   DATA[2120,25] := 2.0;
   DATA[2120,26] := 7.873174;
   DATA[2120,27] := 144.322;
   DATA[2120,28] := 262.0161;
   DATA[2120,29] := 12.03538;
   DATA[2120,30] := 1.726096;
   DATA[2120,31] := 1.28372;
   DATA[2120,32] := 0.7353967;
   DATA[2120,33] := 0.3084265;
   DATA[2120,34] := 2.0;
   DATA[2120,35] := 250.1122;
   DATA[2120,36] := 1.69801;
   DATA[2120,37] := 189.0381;
   DATA[2120,38] := 0.000128152;
   DATA[2120,39] := 1.0;
   DATA[2120,40] := 1.0;
   DATA[2121,0] := 2.573103;
   DATA[2121,1] := 862.3046;
   DATA[2121,2] := 2.0;
   DATA[2121,3] := 2.0;
   DATA[2121,4] := 262.4007;
   DATA[2121,5] := 8.392271;
   DATA[2121,6] := 330.7357;
   DATA[2121,7] := 2.461667;
   DATA[2121,8] := 2.0;
   DATA[2121,9] := 2.0;
   DATA[2121,10] := 2.0;
   DATA[2121,11] := 19.72598;
   DATA[2121,12] := 2.209013;
   DATA[2121,13] := 806.564;
   DATA[2121,14] := 1.0;
   DATA[2121,15] := 2.0;
   DATA[2121,16] := 1.0;
   DATA[2121,17] := 1.0;
   DATA[2121,18] := 1.0;
   DATA[2121,19] := 2.0;
   DATA[2121,20] := 148.808;
   DATA[2121,21] := 154.8065;
   DATA[2121,22] := 1.717489;
   DATA[2121,23] := 839.131;
   DATA[2121,24] := 2.0;
   DATA[2121,25] := 2.0;
   DATA[2121,26] := 7.873174;
   DATA[2121,27] := 144.322;
   DATA[2121,28] := 262.0161;
   DATA[2121,29] := 12.03538;
   DATA[2121,30] := 1.725968;
   DATA[2121,31] := 1.300884;
   DATA[2121,32] := 0.7353967;
   DATA[2121,33] := 0.3084265;
   DATA[2121,34] := 2.0;
   DATA[2121,35] := 250.1122;
   DATA[2121,36] := 1.69801;
   DATA[2121,37] := 189.0381;
   DATA[2121,38] := 0.000128152;
   DATA[2121,39] := 1.0;
   DATA[2121,40] := 1.0;
   DATA[2122,0] := 2.608013;
   DATA[2122,1] := 862.6971;
   DATA[2122,2] := 2.0;
   DATA[2122,3] := 2.0;
   DATA[2122,4] := 262.4007;
   DATA[2122,5] := 8.392271;
   DATA[2122,6] := 330.7357;
   DATA[2122,7] := 2.461667;
   DATA[2122,8] := 2.0;
   DATA[2122,9] := 2.0;
   DATA[2122,10] := 2.0;
   DATA[2122,11] := 19.67155;
   DATA[2122,12] := 2.209013;
   DATA[2122,13] := 806.3237;
   DATA[2122,14] := 1.0;
   DATA[2122,15] := 2.0;
   DATA[2122,16] := 1.0;
   DATA[2122,17] := 1.0;
   DATA[2122,18] := 1.0;
   DATA[2122,19] := 2.0;
   DATA[2122,20] := 148.808;
   DATA[2122,21] := 154.8065;
   DATA[2122,22] := 1.719156;
   DATA[2122,23] := 839.2463;
   DATA[2122,24] := 2.0;
   DATA[2122,25] := 2.0;
   DATA[2122,26] := 7.873174;
   DATA[2122,27] := 144.322;
   DATA[2122,28] := 262.0161;
   DATA[2122,29] := 12.03538;
   DATA[2122,30] := 1.725968;
   DATA[2122,31] := 1.30178;
   DATA[2122,32] := 0.7353967;
   DATA[2122,33] := 0.3084265;
   DATA[2122,34] := 2.0;
   DATA[2122,35] := 250.3365;
   DATA[2122,36] := 1.69801;
   DATA[2122,37] := 189.0381;
   DATA[2122,38] := 0.000128152;
   DATA[2122,39] := 1.0;
   DATA[2122,40] := 1.0;
   DATA[2123,0] := 2.641322;
   DATA[2123,1] := 862.3831;
   DATA[2123,2] := 2.0;
   DATA[2123,3] := 2.0;
   DATA[2123,4] := 262.4007;
   DATA[2123,5] := 8.392271;
   DATA[2123,6] := 330.787;
   DATA[2123,7] := 2.461667;
   DATA[2123,8] := 2.0;
   DATA[2123,9] := 2.0;
   DATA[2123,10] := 2.0;
   DATA[2123,11] := 19.66835;
   DATA[2123,12] := 2.209013;
   DATA[2123,13] := 806.4038;
   DATA[2123,14] := 1.0;
   DATA[2123,15] := 2.0;
   DATA[2123,16] := 1.0;
   DATA[2123,17] := 1.0;
   DATA[2123,18] := 1.0;
   DATA[2123,19] := 2.0;
   DATA[2123,20] := 148.808;
   DATA[2123,21] := 154.8065;
   DATA[2123,22] := 1.719156;
   DATA[2123,23] := 839.0541;
   DATA[2123,24] := 2.0;
   DATA[2123,25] := 2.0;
   DATA[2123,26] := 7.873174;
   DATA[2123,27] := 144.322;
   DATA[2123,28] := 262.0161;
   DATA[2123,29] := 12.03538;
   DATA[2123,30] := 1.725968;
   DATA[2123,31] := 1.30178;
   DATA[2123,32] := 0.7353967;
   DATA[2123,33] := 0.3084265;
   DATA[2123,34] := 2.0;
   DATA[2123,35] := 250.3365;
   DATA[2123,36] := 1.69801;
   DATA[2123,37] := 189.0381;
   DATA[2123,38] := 0.000128152;
   DATA[2123,39] := 1.0;
   DATA[2123,40] := 1.0;
   DATA[2124,0] := 2.660539;
   DATA[2124,1] := 862.6971;
   DATA[2124,2] := 2.0;
   DATA[2124,3] := 2.0;
   DATA[2124,4] := 262.4007;
   DATA[2124,5] := 8.392271;
   DATA[2124,6] := 330.787;
   DATA[2124,7] := 2.461667;
   DATA[2124,8] := 2.0;
   DATA[2124,9] := 2.0;
   DATA[2124,10] := 2.0;
   DATA[2124,11] := 19.64594;
   DATA[2124,12] := 2.212087;
   DATA[2124,13] := 806.524;
   DATA[2124,14] := 1.0;
   DATA[2124,15] := 2.0;
   DATA[2124,16] := 1.0;
   DATA[2124,17] := 1.0;
   DATA[2124,18] := 1.0;
   DATA[2124,19] := 2.0;
   DATA[2124,20] := 148.808;
   DATA[2124,21] := 154.8065;
   DATA[2124,22] := 1.719156;
   DATA[2124,23] := 839.131;
   DATA[2124,24] := 2.0;
   DATA[2124,25] := 2.0;
   DATA[2124,26] := 7.873174;
   DATA[2124,27] := 144.322;
   DATA[2124,28] := 262.0161;
   DATA[2124,29] := 12.03538;
   DATA[2124,30] := 1.725968;
   DATA[2124,31] := 1.29243;
   DATA[2124,32] := 0.7353967;
   DATA[2124,33] := 0.3084265;
   DATA[2124,34] := 2.0;
   DATA[2124,35] := 250.3365;
   DATA[2124,36] := 1.69801;
   DATA[2124,37] := 189.0861;
   DATA[2124,38] := 0.000128152;
   DATA[2124,39] := 1.0;
   DATA[2124,40] := 1.0;
   DATA[2125,0] := 2.660539;
   DATA[2125,1] := 862.8934;
   DATA[2125,2] := 2.0;
   DATA[2125,3] := 2.0;
   DATA[2125,4] := 262.4007;
   DATA[2125,5] := 8.392271;
   DATA[2125,6] := 330.787;
   DATA[2125,7] := 2.461667;
   DATA[2125,8] := 2.0;
   DATA[2125,9] := 2.0;
   DATA[2125,10] := 2.0;
   DATA[2125,11] := 19.64594;
   DATA[2125,12] := 2.212087;
   DATA[2125,13] := 806.524;
   DATA[2125,14] := 1.0;
   DATA[2125,15] := 2.0;
   DATA[2125,16] := 1.0;
   DATA[2125,17] := 1.0;
   DATA[2125,18] := 1.0;
   DATA[2125,19] := 2.0;
   DATA[2125,20] := 148.808;
   DATA[2125,21] := 154.8065;
   DATA[2125,22] := 1.717874;
   DATA[2125,23] := 839.2079;
   DATA[2125,24] := 2.0;
   DATA[2125,25] := 2.0;
   DATA[2125,26] := 7.874135;
   DATA[2125,27] := 144.322;
   DATA[2125,28] := 262.0161;
   DATA[2125,29] := 12.03538;
   DATA[2125,30] := 1.725968;
   DATA[2125,31] := 1.276419;
   DATA[2125,32] := 0.7353967;
   DATA[2125,33] := 0.3084265;
   DATA[2125,34] := 2.0;
   DATA[2125,35] := 250.3365;
   DATA[2125,36] := 1.69801;
   DATA[2125,37] := 189.1662;
   DATA[2125,38] := 0.000128152;
   DATA[2125,39] := 1.0;
   DATA[2125,40] := 1.0;
   DATA[2126,0] := 2.641642;
   DATA[2126,1] := 863.0897;
   DATA[2126,2] := 2.0;
   DATA[2126,3] := 2.0;
   DATA[2126,4] := 262.4007;
   DATA[2126,5] := 8.392271;
   DATA[2126,6] := 330.8383;
   DATA[2126,7] := 2.461282;
   DATA[2126,8] := 2.0;
   DATA[2126,9] := 2.0;
   DATA[2126,10] := 2.0;
   DATA[2126,11] := 19.64594;
   DATA[2126,12] := 2.212087;
   DATA[2126,13] := 806.6842;
   DATA[2126,14] := 1.0;
   DATA[2126,15] := 2.0;
   DATA[2126,16] := 1.0;
   DATA[2126,17] := 1.0;
   DATA[2126,18] := 1.0;
   DATA[2126,19] := 2.0;
   DATA[2126,20] := 148.808;
   DATA[2126,21] := 154.8065;
   DATA[2126,22] := 1.716849;
   DATA[2126,23] := 839.5924;
   DATA[2126,24] := 2.0;
   DATA[2126,25] := 2.0;
   DATA[2126,26] := 7.874135;
   DATA[2126,27] := 144.322;
   DATA[2126,28] := 262.0161;
   DATA[2126,29] := 12.03538;
   DATA[2126,30] := 1.725968;
   DATA[2126,31] := 1.271295;
   DATA[2126,32] := 0.7353967;
   DATA[2126,33] := 0.3084265;
   DATA[2126,34] := 2.0;
   DATA[2126,35] := 250.3365;
   DATA[2126,36] := 1.69801;
   DATA[2126,37] := 189.1662;
   DATA[2126,38] := 0.000128152;
   DATA[2126,39] := 1.0;
   DATA[2126,40] := 1.0;
   DATA[2127,0] := 2.630433;
   DATA[2127,1] := 862.8934;
   DATA[2127,2] := 2.0;
   DATA[2127,3] := 2.0;
   DATA[2127,4] := 262.4007;
   DATA[2127,5] := 8.392271;
   DATA[2127,6] := 330.8383;
   DATA[2127,7] := 2.458847;
   DATA[2127,8] := 2.0;
   DATA[2127,9] := 2.0;
   DATA[2127,10] := 2.0;
   DATA[2127,11] := 19.70677;
   DATA[2127,12] := 2.212087;
   DATA[2127,13] := 806.2036;
   DATA[2127,14] := 1.0;
   DATA[2127,15] := 2.0;
   DATA[2127,16] := 1.0;
   DATA[2127,17] := 1.0;
   DATA[2127,18] := 1.0;
   DATA[2127,19] := 2.0;
   DATA[2127,20] := 148.808;
   DATA[2127,21] := 154.8065;
   DATA[2127,22] := 1.716849;
   DATA[2127,23] := 839.4771;
   DATA[2127,24] := 2.0;
   DATA[2127,25] := 2.0;
   DATA[2127,26] := 7.874135;
   DATA[2127,27] := 144.322;
   DATA[2127,28] := 262.0161;
   DATA[2127,29] := 12.03538;
   DATA[2127,30] := 1.72789;
   DATA[2127,31] := 1.277443;
   DATA[2127,32] := 0.7353967;
   DATA[2127,33] := 0.3084265;
   DATA[2127,34] := 2.0;
   DATA[2127,35] := 250.3365;
   DATA[2127,36] := 1.69801;
   DATA[2127,37] := 189.1662;
   DATA[2127,38] := 0.000128152;
   DATA[2127,39] := 1.0;
   DATA[2127,40] := 1.0;
   DATA[2128,0] := 2.623387;
   DATA[2128,1] := 863.2859;
   DATA[2128,2] := 2.0;
   DATA[2128,3] := 2.0;
   DATA[2128,4] := 262.4007;
   DATA[2128,5] := 8.392271;
   DATA[2128,6] := 330.8383;
   DATA[2128,7] := 2.458847;
   DATA[2128,8] := 2.0;
   DATA[2128,9] := 2.0;
   DATA[2128,10] := 2.0;
   DATA[2128,11] := 19.70677;
   DATA[2128,12] := 2.210294;
   DATA[2128,13] := 806.524;
   DATA[2128,14] := 1.0;
   DATA[2128,15] := 2.0;
   DATA[2128,16] := 1.0;
   DATA[2128,17] := 1.0;
   DATA[2128,18] := 1.0;
   DATA[2128,19] := 2.0;
   DATA[2128,20] := 148.808;
   DATA[2128,21] := 154.8065;
   DATA[2128,22] := 1.716849;
   DATA[2128,23] := 839.5155;
   DATA[2128,24] := 2.0;
   DATA[2128,25] := 2.0;
   DATA[2128,26] := 7.874135;
   DATA[2128,27] := 144.322;
   DATA[2128,28] := 262.0161;
   DATA[2128,29] := 12.03538;
   DATA[2128,30] := 1.728275;
   DATA[2128,31] := 1.291277;
   DATA[2128,32] := 0.7353967;
   DATA[2128,33] := 0.3084265;
   DATA[2128,34] := 2.0;
   DATA[2128,35] := 250.3365;
   DATA[2128,36] := 1.69801;
   DATA[2128,37] := 189.1662;
   DATA[2128,38] := 0.000128152;
   DATA[2128,39] := 1.0;
   DATA[2128,40] := 1.0;
   DATA[2129,0] := 2.622105;
   DATA[2129,1] := 862.9719;
   DATA[2129,2] := 2.0;
   DATA[2129,3] := 2.0;
   DATA[2129,4] := 262.4007;
   DATA[2129,5] := 8.392271;
   DATA[2129,6] := 330.8383;
   DATA[2129,7] := 2.458078;
   DATA[2129,8] := 2.0;
   DATA[2129,9] := 2.0;
   DATA[2129,10] := 2.0;
   DATA[2129,11] := 19.73558;
   DATA[2129,12] := 2.209269;
   DATA[2129,13] := 805.9232;
   DATA[2129,14] := 1.0;
   DATA[2129,15] := 2.0;
   DATA[2129,16] := 1.0;
   DATA[2129,17] := 1.0;
   DATA[2129,18] := 1.0;
   DATA[2129,19] := 2.0;
   DATA[2129,20] := 148.808;
   DATA[2129,21] := 154.8065;
   DATA[2129,22] := 1.716849;
   DATA[2129,23] := 839.2463;
   DATA[2129,24] := 2.0;
   DATA[2129,25] := 2.0;
   DATA[2129,26] := 7.874135;
   DATA[2129,27] := 144.322;
   DATA[2129,28] := 262.0161;
   DATA[2129,29] := 12.03538;
   DATA[2129,30] := 1.728275;
   DATA[2129,31] := 1.291789;
   DATA[2129,32] := 0.7353967;
   DATA[2129,33] := 0.3084265;
   DATA[2129,34] := 2.0;
   DATA[2129,35] := 250.3365;
   DATA[2129,36] := 1.69801;
   DATA[2129,37] := 189.1662;
   DATA[2129,38] := 0.000128152;
   DATA[2129,39] := 1.0;
   DATA[2129,40] := 1.0;
   DATA[2130,0] := 2.606091;
   DATA[2130,1] := 863.2859;
   DATA[2130,2] := 2.0;
   DATA[2130,3] := 2.0;
   DATA[2130,4] := 262.4007;
   DATA[2130,5] := 8.392271;
   DATA[2130,6] := 330.8383;
   DATA[2130,7] := 2.458078;
   DATA[2130,8] := 2.0;
   DATA[2130,9] := 2.0;
   DATA[2130,10] := 2.0;
   DATA[2130,11] := 19.73558;
   DATA[2130,12] := 2.209269;
   DATA[2130,13] := 805.9232;
   DATA[2130,14] := 1.0;
   DATA[2130,15] := 2.0;
   DATA[2130,16] := 1.0;
   DATA[2130,17] := 1.0;
   DATA[2130,18] := 1.0;
   DATA[2130,19] := 2.0;
   DATA[2130,20] := 148.808;
   DATA[2130,21] := 154.8065;
   DATA[2130,22] := 1.716849;
   DATA[2130,23] := 839.4001;
   DATA[2130,24] := 2.0;
   DATA[2130,25] := 2.0;
   DATA[2130,26] := 7.874135;
   DATA[2130,27] := 144.322;
   DATA[2130,28] := 262.0161;
   DATA[2130,29] := 12.03538;
   DATA[2130,30] := 1.728275;
   DATA[2130,31] := 1.289868;
   DATA[2130,32] := 0.7379573;
   DATA[2130,33] := 0.3084265;
   DATA[2130,34] := 2.0;
   DATA[2130,35] := 250.3365;
   DATA[2130,36] := 1.69801;
   DATA[2130,37] := 189.1662;
   DATA[2130,38] := 0.000128152;
   DATA[2130,39] := 1.0;
   DATA[2130,40] := 1.0;
   DATA[2131,0] := 2.587195;
   DATA[2131,1] := 863.5999;
   DATA[2131,2] := 2.0;
   DATA[2131,3] := 2.0;
   DATA[2131,4] := 262.4007;
   DATA[2131,5] := 8.392271;
   DATA[2131,6] := 330.8383;
   DATA[2131,7] := 2.458078;
   DATA[2131,8] := 2.0;
   DATA[2131,9] := 2.0;
   DATA[2131,10] := 2.0;
   DATA[2131,11] := 19.77079;
   DATA[2131,12] := 2.209269;
   DATA[2131,13] := 805.7229;
   DATA[2131,14] := 1.0;
   DATA[2131,15] := 2.0;
   DATA[2131,16] := 1.0;
   DATA[2131,17] := 1.0;
   DATA[2131,18] := 1.0;
   DATA[2131,19] := 2.0;
   DATA[2131,20] := 148.808;
   DATA[2131,21] := 154.8065;
   DATA[2131,22] := 1.716849;
   DATA[2131,23] := 839.0541;
   DATA[2131,24] := 2.0;
   DATA[2131,25] := 2.0;
   DATA[2131,26] := 7.874135;
   DATA[2131,27] := 144.322;
   DATA[2131,28] := 262.0161;
   DATA[2131,29] := 12.03538;
   DATA[2131,30] := 1.726096;
   DATA[2131,31] := 1.269117;
   DATA[2131,32] := 0.7379573;
   DATA[2131,33] := 0.3084265;
   DATA[2131,34] := 2.0;
   DATA[2131,35] := 250.3365;
   DATA[2131,36] := 1.69801;
   DATA[2131,37] := 189.1662;
   DATA[2131,38] := 0.000128152;
   DATA[2131,39] := 1.0;
   DATA[2131,40] := 1.0;
   DATA[2132,0] := 2.567338;
   DATA[2132,1] := 863.4822;
   DATA[2132,2] := 2.0;
   DATA[2132,3] := 2.0;
   DATA[2132,4] := 262.4007;
   DATA[2132,5] := 8.392271;
   DATA[2132,6] := 330.8383;
   DATA[2132,7] := 2.458078;
   DATA[2132,8] := 2.0;
   DATA[2132,9] := 2.0;
   DATA[2132,10] := 2.0;
   DATA[2132,11] := 19.77079;
   DATA[2132,12] := 2.209269;
   DATA[2132,13] := 805.8831;
   DATA[2132,14] := 1.0;
   DATA[2132,15] := 2.0;
   DATA[2132,16] := 1.0;
   DATA[2132,17] := 1.0;
   DATA[2132,18] := 1.0;
   DATA[2132,19] := 2.0;
   DATA[2132,20] := 148.808;
   DATA[2132,21] := 154.8065;
   DATA[2132,22] := 1.717746;
   DATA[2132,23] := 839.3232;
   DATA[2132,24] := 2.0;
   DATA[2132,25] := 2.0;
   DATA[2132,26] := 7.874135;
   DATA[2132,27] := 144.322;
   DATA[2132,28] := 262.0161;
   DATA[2132,29] := 12.03538;
   DATA[2132,30] := 1.726096;
   DATA[2132,31] := 1.265659;
   DATA[2132,32] := 0.7379573;
   DATA[2132,33] := 0.3084265;
   DATA[2132,34] := 2.0;
   DATA[2132,35] := 250.4326;
   DATA[2132,36] := 1.69801;
   DATA[2132,37] := 189.1662;
   DATA[2132,38] := 0.000128152;
   DATA[2132,39] := 1.0;
   DATA[2132,40] := 1.0;
   DATA[2133,0] := 2.558691;
   DATA[2133,1] := 863.8354;
   DATA[2133,2] := 2.0;
   DATA[2133,3] := 2.0;
   DATA[2133,4] := 262.4007;
   DATA[2133,5] := 8.392271;
   DATA[2133,6] := 330.8383;
   DATA[2133,7] := 2.458078;
   DATA[2133,8] := 2.0;
   DATA[2133,9] := 2.0;
   DATA[2133,10] := 2.0;
   DATA[2133,11] := 19.77079;
   DATA[2133,12] := 2.209269;
   DATA[2133,13] := 805.7229;
   DATA[2133,14] := 1.0;
   DATA[2133,15] := 2.0;
   DATA[2133,16] := 1.0;
   DATA[2133,17] := 1.0;
   DATA[2133,18] := 1.0;
   DATA[2133,19] := 2.0;
   DATA[2133,20] := 148.808;
   DATA[2133,21] := 154.9603;
   DATA[2133,22] := 1.718771;
   DATA[2133,23] := 839.0541;
   DATA[2133,24] := 2.0;
   DATA[2133,25] := 2.0;
   DATA[2133,26] := 7.874135;
   DATA[2133,27] := 144.322;
   DATA[2133,28] := 262.0161;
   DATA[2133,29] := 12.03538;
   DATA[2133,30] := 1.726096;
   DATA[2133,31] := 1.280902;
   DATA[2133,32] := 0.7366771;
   DATA[2133,33] := 0.3070813;
   DATA[2133,34] := 2.0;
   DATA[2133,35] := 250.4967;
   DATA[2133,36] := 1.69801;
   DATA[2133,37] := 189.1662;
   DATA[2133,38] := 0.000128152;
   DATA[2133,39] := 1.0;
   DATA[2133,40] := 1.0;
   DATA[2134,0] := 2.535951;
   DATA[2134,1] := 863.7962;
   DATA[2134,2] := 2.0;
   DATA[2134,3] := 2.0;
   DATA[2134,4] := 262.4007;
   DATA[2134,5] := 8.392271;
   DATA[2134,6] := 330.8383;
   DATA[2134,7] := 2.458078;
   DATA[2134,8] := 2.0;
   DATA[2134,9] := 2.0;
   DATA[2134,10] := 2.0;
   DATA[2134,11] := 19.77079;
   DATA[2134,12] := 2.209269;
   DATA[2134,13] := 805.6829;
   DATA[2134,14] := 1.0;
   DATA[2134,15] := 2.0;
   DATA[2134,16] := 1.0;
   DATA[2134,17] := 1.0;
   DATA[2134,18] := 1.0;
   DATA[2134,19] := 2.0;
   DATA[2134,20] := 148.808;
   DATA[2134,21] := 154.9603;
   DATA[2134,22] := 1.718771;
   DATA[2134,23] := 839.2463;
   DATA[2134,24] := 2.0;
   DATA[2134,25] := 2.0;
   DATA[2134,26] := 7.874135;
   DATA[2134,27] := 144.322;
   DATA[2134,28] := 262.0161;
   DATA[2134,29] := 12.03538;
   DATA[2134,30] := 1.726096;
   DATA[2134,31] := 1.280005;
   DATA[2134,32] := 0.7359089;
   DATA[2134,33] := 0.3070813;
   DATA[2134,34] := 2.0;
   DATA[2134,35] := 250.4967;
   DATA[2134,36] := 1.69801;
   DATA[2134,37] := 189.1662;
   DATA[2134,38] := 0.000128152;
   DATA[2134,39] := 1.0;
   DATA[2134,40] := 1.0;
   DATA[2135,0] := 2.520257;
   DATA[2135,1] := 864.1887;
   DATA[2135,2] := 2.0;
   DATA[2135,3] := 2.0;
   DATA[2135,4] := 262.4007;
   DATA[2135,5] := 8.392271;
   DATA[2135,6] := 330.8383;
   DATA[2135,7] := 2.459744;
   DATA[2135,8] := 2.0;
   DATA[2135,9] := 2.0;
   DATA[2135,10] := 2.0;
   DATA[2135,11] := 19.73238;
   DATA[2135,12] := 2.209269;
   DATA[2135,13] := 805.5627;
   DATA[2135,14] := 1.0;
   DATA[2135,15] := 2.0;
   DATA[2135,16] := 1.0;
   DATA[2135,17] := 1.0;
   DATA[2135,18] := 1.0;
   DATA[2135,19] := 2.0;
   DATA[2135,20] := 148.808;
   DATA[2135,21] := 154.9603;
   DATA[2135,22] := 1.720309;
   DATA[2135,23] := 838.8234;
   DATA[2135,24] := 2.0;
   DATA[2135,25] := 2.0;
   DATA[2135,26] := 7.874135;
   DATA[2135,27] := 144.322;
   DATA[2135,28] := 262.0161;
   DATA[2135,29] := 12.03538;
   DATA[2135,30] := 1.726096;
   DATA[2135,31] := 1.275778;
   DATA[2135,32] := 0.7348846;
   DATA[2135,33] := 0.3075297;
   DATA[2135,34] := 2.0;
   DATA[2135,35] := 250.4967;
   DATA[2135,36] := 1.69801;
   DATA[2135,37] := 189.2143;
   DATA[2135,38] := 0.000128152;
   DATA[2135,39] := 1.0;
   DATA[2135,40] := 1.0;
   DATA[2136,0] := 2.502642;
   DATA[2136,1] := 864.385;
   DATA[2136,2] := 2.0;
   DATA[2136,3] := 2.0;
   DATA[2136,4] := 262.4007;
   DATA[2136,5] := 8.392271;
   DATA[2136,6] := 330.8383;
   DATA[2136,7] := 2.459744;
   DATA[2136,8] := 2.0;
   DATA[2136,9] := 2.0;
   DATA[2136,10] := 2.0;
   DATA[2136,11] := 19.73238;
   DATA[2136,12] := 2.209269;
   DATA[2136,13] := 805.4025;
   DATA[2136,14] := 1.0;
   DATA[2136,15] := 2.0;
   DATA[2136,16] := 1.0;
   DATA[2136,17] := 1.0;
   DATA[2136,18] := 1.0;
   DATA[2136,19] := 2.0;
   DATA[2136,20] := 148.808;
   DATA[2136,21] := 154.9603;
   DATA[2136,22] := 1.720309;
   DATA[2136,23] := 838.6311;
   DATA[2136,24] := 2.0;
   DATA[2136,25] := 2.0;
   DATA[2136,26] := 7.874135;
   DATA[2136,27] := 144.322;
   DATA[2136,28] := 262.0161;
   DATA[2136,29] := 12.03538;
   DATA[2136,30] := 1.726096;
   DATA[2136,31] := 1.276419;
   DATA[2136,32] := 0.7348846;
   DATA[2136,33] := 0.3083624;
   DATA[2136,34] := 2.0;
   DATA[2136,35] := 250.4967;
   DATA[2136,36] := 1.69801;
   DATA[2136,37] := 189.3585;
   DATA[2136,38] := 0.000128152;
   DATA[2136,39] := 1.0;
   DATA[2136,40] := 1.0;
   DATA[2137,0] := 2.48823;
   DATA[2137,1] := 864.6205;
   DATA[2137,2] := 2.0;
   DATA[2137,3] := 2.0;
   DATA[2137,4] := 262.4007;
   DATA[2137,5] := 8.392271;
   DATA[2137,6] := 330.8126;
   DATA[2137,7] := 2.460129;
   DATA[2137,8] := 2.0;
   DATA[2137,9] := 2.0;
   DATA[2137,10] := 2.0;
   DATA[2137,11] := 19.73238;
   DATA[2137,12] := 2.209269;
   DATA[2137,13] := 805.2022;
   DATA[2137,14] := 1.0;
   DATA[2137,15] := 2.0;
   DATA[2137,16] := 1.0;
   DATA[2137,17] := 1.0;
   DATA[2137,18] := 1.0;
   DATA[2137,19] := 2.0;
   DATA[2137,20] := 148.808;
   DATA[2137,21] := 154.9603;
   DATA[2137,22] := 1.720309;
   DATA[2137,23] := 838.0928;
   DATA[2137,24] := 2.0;
   DATA[2137,25] := 2.0;
   DATA[2137,26] := 7.874135;
   DATA[2137,27] := 144.322;
   DATA[2137,28] := 262.0161;
   DATA[2137,29] := 12.03538;
   DATA[2137,30] := 1.728019;
   DATA[2137,31] := 1.270398;
   DATA[2137,32] := 0.7348846;
   DATA[2137,33] := 0.3075937;
   DATA[2137,34] := 2.0;
   DATA[2137,35] := 250.4967;
   DATA[2137,36] := 1.69801;
   DATA[2137,37] := 189.3585;
   DATA[2137,38] := 0.000128152;
   DATA[2137,39] := 1.0;
   DATA[2137,40] := 1.0;
   DATA[2138,0] := 2.467092;
   DATA[2138,1] := 864.8168;
   DATA[2138,2] := 2.0;
   DATA[2138,3] := 2.0;
   DATA[2138,4] := 262.4007;
   DATA[2138,5] := 8.392271;
   DATA[2138,6] := 330.6075;
   DATA[2138,7] := 2.460129;
   DATA[2138,8] := 2.0;
   DATA[2138,9] := 2.0;
   DATA[2138,10] := 2.0;
   DATA[2138,11] := 19.73238;
   DATA[2138,12] := 2.210037;
   DATA[2138,13] := 805.3224;
   DATA[2138,14] := 1.0;
   DATA[2138,15] := 2.0;
   DATA[2138,16] := 1.0;
   DATA[2138,17] := 1.0;
   DATA[2138,18] := 1.0;
   DATA[2138,19] := 2.0;
   DATA[2138,20] := 148.808;
   DATA[2138,21] := 154.9603;
   DATA[2138,22] := 1.720309;
   DATA[2138,23] := 838.1312;
   DATA[2138,24] := 2.0;
   DATA[2138,25] := 2.0;
   DATA[2138,26] := 7.874135;
   DATA[2138,27] := 144.322;
   DATA[2138,28] := 262.0161;
   DATA[2138,29] := 12.03538;
   DATA[2138,30] := 1.728788;
   DATA[2138,31] := 1.278468;
   DATA[2138,32] := 0.7348846;
   DATA[2138,33] := 0.3069532;
   DATA[2138,34] := 2.0;
   DATA[2138,35] := 250.4967;
   DATA[2138,36] := 1.69801;
   DATA[2138,37] := 189.3585;
   DATA[2138,38] := 0.000128152;
   DATA[2138,39] := 1.0;
   DATA[2138,40] := 1.0;
   DATA[2139,0] := 2.458764;
   DATA[2139,1] := 864.6597;
   DATA[2139,2] := 2.0;
   DATA[2139,3] := 2.0;
   DATA[2139,4] := 262.4007;
   DATA[2139,5] := 8.392271;
   DATA[2139,6] := 330.6075;
   DATA[2139,7] := 2.460129;
   DATA[2139,8] := 2.0;
   DATA[2139,9] := 2.0;
   DATA[2139,10] := 2.0;
   DATA[2139,11] := 19.73238;
   DATA[2139,12] := 2.21055;
   DATA[2139,13] := 805.2022;
   DATA[2139,14] := 1.0;
   DATA[2139,15] := 2.0;
   DATA[2139,16] := 1.0;
   DATA[2139,17] := 1.0;
   DATA[2139,18] := 1.0;
   DATA[2139,19] := 2.0;
   DATA[2139,20] := 148.808;
   DATA[2139,21] := 155.0884;
   DATA[2139,22] := 1.720309;
   DATA[2139,23] := 838.0928;
   DATA[2139,24] := 2.0;
   DATA[2139,25] := 2.0;
   DATA[2139,26] := 7.874135;
   DATA[2139,27] := 144.322;
   DATA[2139,28] := 262.0161;
   DATA[2139,29] := 12.03538;
   DATA[2139,30] := 1.728788;
   DATA[2139,31] := 1.296016;
   DATA[2139,32] := 0.7348846;
   DATA[2139,33] := 0.3065048;
   DATA[2139,34] := 2.0;
   DATA[2139,35] := 250.4967;
   DATA[2139,36] := 1.69801;
   DATA[2139,37] := 189.3585;
   DATA[2139,38] := 0.000128152;
   DATA[2139,39] := 1.0;
   DATA[2139,40] := 1.0;
   DATA[2140,0] := 2.436665;
   DATA[2140,1] := 864.4635;
   DATA[2140,2] := 2.0;
   DATA[2140,3] := 2.0;
   DATA[2140,4] := 262.4007;
   DATA[2140,5] := 8.392271;
   DATA[2140,6] := 330.6075;
   DATA[2140,7] := 2.460641;
   DATA[2140,8] := 2.0;
   DATA[2140,9] := 2.0;
   DATA[2140,10] := 2.0;
   DATA[2140,11] := 19.7836;
   DATA[2140,12] := 2.21055;
   DATA[2140,13] := 804.6815;
   DATA[2140,14] := 1.0;
   DATA[2140,15] := 2.0;
   DATA[2140,16] := 1.0;
   DATA[2140,17] := 1.0;
   DATA[2140,18] := 1.0;
   DATA[2140,19] := 2.0;
   DATA[2140,20] := 148.808;
   DATA[2140,21] := 155.0884;
   DATA[2140,22] := 1.720309;
   DATA[2140,23] := 837.7852;
   DATA[2140,24] := 2.0;
   DATA[2140,25] := 2.0;
   DATA[2140,26] := 7.874135;
   DATA[2140,27] := 144.322;
   DATA[2140,28] := 262.0161;
   DATA[2140,29] := 12.03538;
   DATA[2140,30] := 1.728788;
   DATA[2140,31] := 1.310747;
   DATA[2140,32] := 0.7348846;
   DATA[2140,33] := 0.3065048;
   DATA[2140,34] := 2.0;
   DATA[2140,35] := 250.4967;
   DATA[2140,36] := 1.69801;
   DATA[2140,37] := 189.2464;
   DATA[2140,38] := 0.000128152;
   DATA[2140,39] := 1.0;
   DATA[2140,40] := 1.0;
   DATA[2141,0] := 2.428018;
   DATA[2141,1] := 864.228;
   DATA[2141,2] := 2.0;
   DATA[2141,3] := 2.0;
   DATA[2141,4] := 262.4007;
   DATA[2141,5] := 8.392271;
   DATA[2141,6] := 330.6075;
   DATA[2141,7] := 2.462564;
   DATA[2141,8] := 2.0;
   DATA[2141,9] := 2.0;
   DATA[2141,10] := 2.0;
   DATA[2141,11] := 19.7836;
   DATA[2141,12] := 2.21055;
   DATA[2141,13] := 804.6014;
   DATA[2141,14] := 1.0;
   DATA[2141,15] := 2.0;
   DATA[2141,16] := 1.0;
   DATA[2141,17] := 1.0;
   DATA[2141,18] := 1.0;
   DATA[2141,19] := 2.0;
   DATA[2141,20] := 148.808;
   DATA[2141,21] := 155.0884;
   DATA[2141,22] := 1.716464;
   DATA[2141,23] := 838.0543;
   DATA[2141,24] := 2.0;
   DATA[2141,25] := 2.0;
   DATA[2141,26] := 7.874135;
   DATA[2141,27] := 144.322;
   DATA[2141,28] := 262.0161;
   DATA[2141,29] := 12.03538;
   DATA[2141,30] := 1.728788;
   DATA[2141,31] := 1.312284;
   DATA[2141,32] := 0.7348846;
   DATA[2141,33] := 0.3065048;
   DATA[2141,34] := 2.0;
   DATA[2141,35] := 250.4967;
   DATA[2141,36] := 1.69801;
   DATA[2141,37] := 189.2464;
   DATA[2141,38] := 0.000128152;
   DATA[2141,39] := 1.0;
   DATA[2141,40] := 1.0;
   DATA[2142,0] := 2.428018;
   DATA[2142,1] := 864.2672;
   DATA[2142,2] := 2.0;
   DATA[2142,3] := 2.0;
   DATA[2142,4] := 262.4007;
   DATA[2142,5] := 8.392271;
   DATA[2142,6] := 330.6075;
   DATA[2142,7] := 2.463845;
   DATA[2142,8] := 2.0;
   DATA[2142,9] := 2.0;
   DATA[2142,10] := 2.0;
   DATA[2142,11] := 19.7836;
   DATA[2142,12] := 2.209525;
   DATA[2142,13] := 804.8017;
   DATA[2142,14] := 1.0;
   DATA[2142,15] := 2.0;
   DATA[2142,16] := 1.0;
   DATA[2142,17] := 1.0;
   DATA[2142,18] := 1.0;
   DATA[2142,19] := 2.0;
   DATA[2142,20] := 148.808;
   DATA[2142,21] := 155.0884;
   DATA[2142,22] := 1.716464;
   DATA[2142,23] := 838.4773;
   DATA[2142,24] := 2.0;
   DATA[2142,25] := 2.0;
   DATA[2142,26] := 7.874135;
   DATA[2142,27] := 144.1938;
   DATA[2142,28] := 262.0161;
   DATA[2142,29] := 12.03538;
   DATA[2142,30] := 1.728788;
   DATA[2142,31] := 1.308569;
   DATA[2142,32] := 0.7348846;
   DATA[2142,33] := 0.3065048;
   DATA[2142,34] := 2.0;
   DATA[2142,35] := 250.3525;
   DATA[2142,36] := 1.69801;
   DATA[2142,37] := 189.2464;
   DATA[2142,38] := 0.000128152;
   DATA[2142,39] := 1.0;
   DATA[2142,40] := 1.0;
   DATA[2143,0] := 2.43058;
   DATA[2143,1] := 864.385;
   DATA[2143,2] := 2.0;
   DATA[2143,3] := 2.0;
   DATA[2143,4] := 262.4007;
   DATA[2143,5] := 8.392271;
   DATA[2143,6] := 330.6075;
   DATA[2143,7] := 2.463845;
   DATA[2143,8] := 2.0;
   DATA[2143,9] := 2.0;
   DATA[2143,10] := 2.0;
   DATA[2143,11] := 19.7836;
   DATA[2143,12] := 2.209397;
   DATA[2143,13] := 804.5613;
   DATA[2143,14] := 1.0;
   DATA[2143,15] := 2.0;
   DATA[2143,16] := 1.0;
   DATA[2143,17] := 1.0;
   DATA[2143,18] := 1.0;
   DATA[2143,19] := 2.0;
   DATA[2143,20] := 148.808;
   DATA[2143,21] := 155.0884;
   DATA[2143,22] := 1.716464;
   DATA[2143,23] := 838.6311;
   DATA[2143,24] := 2.0;
   DATA[2143,25] := 2.0;
   DATA[2143,26] := 7.874135;
   DATA[2143,27] := 144.1938;
   DATA[2143,28] := 262.0161;
   DATA[2143,29] := 12.03538;
   DATA[2143,30] := 1.726737;
   DATA[2143,31] := 1.288715;
   DATA[2143,32] := 0.7348846;
   DATA[2143,33] := 0.3065048;
   DATA[2143,34] := 2.0;
   DATA[2143,35] := 250.3525;
   DATA[2143,36] := 1.69801;
   DATA[2143,37] := 189.2464;
   DATA[2143,38] := 0.000128152;
   DATA[2143,39] := 1.0;
   DATA[2143,40] := 1.0;
   DATA[2144,0] := 2.466771;
   DATA[2144,1] := 864.2672;
   DATA[2144,2] := 2.0;
   DATA[2144,3] := 2.0;
   DATA[2144,4] := 262.4007;
   DATA[2144,5] := 8.392271;
   DATA[2144,6] := 330.6075;
   DATA[2144,7] := 2.462564;
   DATA[2144,8] := 2.0;
   DATA[2144,9] := 2.0;
   DATA[2144,10] := 2.0;
   DATA[2144,11] := 19.64594;
   DATA[2144,12] := 2.209397;
   DATA[2144,13] := 804.8017;
   DATA[2144,14] := 1.0;
   DATA[2144,15] := 2.0;
   DATA[2144,16] := 1.0;
   DATA[2144,17] := 1.0;
   DATA[2144,18] := 1.0;
   DATA[2144,19] := 2.0;
   DATA[2144,20] := 148.808;
   DATA[2144,21] := 155.0884;
   DATA[2144,22] := 1.713261;
   DATA[2144,23] := 839.0925;
   DATA[2144,24] := 2.0;
   DATA[2144,25] := 2.0;
   DATA[2144,26] := 7.874135;
   DATA[2144,27] := 144.1938;
   DATA[2144,28] := 262.0161;
   DATA[2144,29] := 12.03538;
   DATA[2144,30] := 1.72507;
   DATA[2144,31] := 1.281927;
   DATA[2144,32] := 0.7348846;
   DATA[2144,33] := 0.3065048;
   DATA[2144,34] := 2.0;
   DATA[2144,35] := 250.3525;
   DATA[2144,36] := 1.69801;
   DATA[2144,37] := 188.974;
   DATA[2144,38] := 0.000128152;
   DATA[2144,39] := 1.0;
   DATA[2144,40] := 1.0;
   DATA[2145,0] := 2.513532;
   DATA[2145,1] := 864.071;
   DATA[2145,2] := 2.0;
   DATA[2145,3] := 2.0;
   DATA[2145,4] := 262.4007;
   DATA[2145,5] := 8.392271;
   DATA[2145,6] := 330.6075;
   DATA[2145,7] := 2.462179;
   DATA[2145,8] := 2.0;
   DATA[2145,9] := 2.0;
   DATA[2145,10] := 2.0;
   DATA[2145,11] := 19.56591;
   DATA[2145,12] := 2.209397;
   DATA[2145,13] := 805.002;
   DATA[2145,14] := 1.0;
   DATA[2145,15] := 2.0;
   DATA[2145,16] := 1.0;
   DATA[2145,17] := 1.0;
   DATA[2145,18] := 1.0;
   DATA[2145,19] := 2.0;
   DATA[2145,20] := 148.808;
   DATA[2145,21] := 155.0884;
   DATA[2145,22] := 1.713261;
   DATA[2145,23] := 838.9387;
   DATA[2145,24] := 2.0;
   DATA[2145,25] := 2.0;
   DATA[2145,26] := 7.874135;
   DATA[2145,27] := 144.1938;
   DATA[2145,28] := 262.0161;
   DATA[2145,29] := 12.03538;
   DATA[2145,30] := 1.72507;
   DATA[2145,31] := 1.271935;
   DATA[2145,32] := 0.7353967;
   DATA[2145,33] := 0.3065048;
   DATA[2145,34] := 2.0;
   DATA[2145,35] := 250.2403;
   DATA[2145,36] := 1.69801;
   DATA[2145,37] := 188.974;
   DATA[2145,38] := 0.000128152;
   DATA[2145,39] := 1.0;
   DATA[2145,40] := 1.0;
   DATA[2146,0] := 2.550364;
   DATA[2146,1] := 863.8354;
   DATA[2146,2] := 2.0;
   DATA[2146,3] := 2.0;
   DATA[2146,4] := 262.4007;
   DATA[2146,5] := 8.392271;
   DATA[2146,6] := 330.6075;
   DATA[2146,7] := 2.461667;
   DATA[2146,8] := 2.0;
   DATA[2146,9] := 2.0;
   DATA[2146,10] := 2.0;
   DATA[2146,11] := 19.50829;
   DATA[2146,12] := 2.209397;
   DATA[2146,13] := 805.5226;
   DATA[2146,14] := 1.0;
   DATA[2146,15] := 2.0;
   DATA[2146,16] := 1.0;
   DATA[2146,17] := 1.0;
   DATA[2146,18] := 1.0;
   DATA[2146,19] := 2.0;
   DATA[2146,20] := 148.808;
   DATA[2146,21] := 155.0884;
   DATA[2146,22] := 1.713261;
   DATA[2146,23] := 839.4771;
   DATA[2146,24] := 2.0;
   DATA[2146,25] := 2.0;
   DATA[2146,26] := 7.874135;
   DATA[2146,27] := 144.1938;
   DATA[2146,28] := 262.0161;
   DATA[2146,29] := 12.03538;
   DATA[2146,30] := 1.72507;
   DATA[2146,31] := 1.271679;
   DATA[2146,32] := 0.7353967;
   DATA[2146,33] := 0.3084905;
   DATA[2146,34] := 2.0;
   DATA[2146,35] := 250.016;
   DATA[2146,36] := 1.69801;
   DATA[2146,37] := 188.974;
   DATA[2146,38] := 0.000128152;
   DATA[2146,39] := 1.0;
   DATA[2146,40] := 1.0;
   DATA[2147,0] := 2.596163;
   DATA[2147,1] := 863.7962;
   DATA[2147,2] := 2.0;
   DATA[2147,3] := 2.0;
   DATA[2147,4] := 262.4007;
   DATA[2147,5] := 8.392271;
   DATA[2147,6] := 330.6075;
   DATA[2147,7] := 2.461667;
   DATA[2147,8] := 2.0;
   DATA[2147,9] := 2.0;
   DATA[2147,10] := 2.0;
   DATA[2147,11] := 19.50829;
   DATA[2147,12] := 2.209397;
   DATA[2147,13] := 805.5627;
   DATA[2147,14] := 1.0;
   DATA[2147,15] := 2.0;
   DATA[2147,16] := 1.0;
   DATA[2147,17] := 1.0;
   DATA[2147,18] := 1.0;
   DATA[2147,19] := 2.0;
   DATA[2147,20] := 148.808;
   DATA[2147,21] := 155.0884;
   DATA[2147,22] := 1.713261;
   DATA[2147,23] := 839.4386;
   DATA[2147,24] := 2.0;
   DATA[2147,25] := 2.0;
   DATA[2147,26] := 7.874135;
   DATA[2147,27] := 144.1938;
   DATA[2147,28] := 262.0161;
   DATA[2147,29] := 12.03538;
   DATA[2147,30] := 1.724301;
   DATA[2147,31] := 1.279877;
   DATA[2147,32] := 0.7353967;
   DATA[2147,33] := 0.3072094;
   DATA[2147,34] := 2.0;
   DATA[2147,35] := 250.0;
   DATA[2147,36] := 1.69801;
   DATA[2147,37] := 188.8138;
   DATA[2147,38] := 0.000128152;
   DATA[2147,39] := 1.0;
   DATA[2147,40] := 1.0;
   DATA[2148,0] := 2.62723;
   DATA[2148,1] := 863.8747;
   DATA[2148,2] := 2.0;
   DATA[2148,3] := 2.0;
   DATA[2148,4] := 262.4007;
   DATA[2148,5] := 8.392271;
   DATA[2148,6] := 330.6075;
   DATA[2148,7] := 2.461667;
   DATA[2148,8] := 2.0;
   DATA[2148,9] := 2.0;
   DATA[2148,10] := 2.0;
   DATA[2148,11] := 19.57872;
   DATA[2148,12] := 2.209397;
   DATA[2148,13] := 805.9232;
   DATA[2148,14] := 1.0;
   DATA[2148,15] := 2.0;
   DATA[2148,16] := 1.0;
   DATA[2148,17] := 1.0;
   DATA[2148,18] := 1.0;
   DATA[2148,19] := 2.0;
   DATA[2148,20] := 148.808;
   DATA[2148,21] := 155.0884;
   DATA[2148,22] := 1.713261;
   DATA[2148,23] := 839.9769;
   DATA[2148,24] := 2.0;
   DATA[2148,25] := 2.0;
   DATA[2148,26] := 7.874135;
   DATA[2148,27] := 144.1938;
   DATA[2148,28] := 262.0161;
   DATA[2148,29] := 12.03538;
   DATA[2148,30] := 1.723661;
   DATA[2148,31] := 1.283079;
   DATA[2148,32] := 0.7353967;
   DATA[2148,33] := 0.3065689;
   DATA[2148,34] := 2.0;
   DATA[2148,35] := 250.0;
   DATA[2148,36] := 1.69801;
   DATA[2148,37] := 188.8138;
   DATA[2148,38] := 0.000128152;
   DATA[2148,39] := 1.0;
   DATA[2148,40] := 1.0;
   DATA[2149,0] := 2.647407;
   DATA[2149,1] := 863.8747;
   DATA[2149,2] := 2.0;
   DATA[2149,3] := 2.0;
   DATA[2149,4] := 262.4007;
   DATA[2149,5] := 8.392271;
   DATA[2149,6] := 330.6075;
   DATA[2149,7] := 2.461667;
   DATA[2149,8] := 2.0;
   DATA[2149,9] := 2.0;
   DATA[2149,10] := 2.0;
   DATA[2149,11] := 19.61393;
   DATA[2149,12] := 2.209397;
   DATA[2149,13] := 806.1235;
   DATA[2149,14] := 1.0;
   DATA[2149,15] := 2.0;
   DATA[2149,16] := 1.0;
   DATA[2149,17] := 1.0;
   DATA[2149,18] := 1.0;
   DATA[2149,19] := 2.0;
   DATA[2149,20] := 148.808;
   DATA[2149,21] := 155.0884;
   DATA[2149,22] := 1.713261;
   DATA[2149,23] := 840.2845;
   DATA[2149,24] := 2.0;
   DATA[2149,25] := 2.0;
   DATA[2149,26] := 7.874135;
   DATA[2149,27] := 144.1938;
   DATA[2149,28] := 262.0161;
   DATA[2149,29] := 12.03538;
   DATA[2149,30] := 1.723661;
   DATA[2149,31] := 1.291405;
   DATA[2149,32] := 0.7353967;
   DATA[2149,33] := 0.3084265;
   DATA[2149,34] := 2.0;
   DATA[2149,35] := 250.0;
   DATA[2149,36] := 1.69801;
   DATA[2149,37] := 188.8138;
   DATA[2149,38] := 0.000128152;
   DATA[2149,39] := 1.0;
   DATA[2149,40] := 1.0;
   DATA[2150,0] := 2.659578;
   DATA[2150,1] := 863.4822;
   DATA[2150,2] := 2.0;
   DATA[2150,3] := 2.0;
   DATA[2150,4] := 262.4007;
   DATA[2150,5] := 8.392271;
   DATA[2150,6] := 330.6075;
   DATA[2150,7] := 2.461667;
   DATA[2150,8] := 2.0;
   DATA[2150,9] := 2.0;
   DATA[2150,10] := 2.0;
   DATA[2150,11] := 19.61393;
   DATA[2150,12] := 2.209397;
   DATA[2150,13] := 806.2036;
   DATA[2150,14] := 1.0;
   DATA[2150,15] := 2.0;
   DATA[2150,16] := 1.0;
   DATA[2150,17] := 1.0;
   DATA[2150,18] := 1.0;
   DATA[2150,19] := 2.0;
   DATA[2150,20] := 148.808;
   DATA[2150,21] := 155.0884;
   DATA[2150,22] := 1.712363;
   DATA[2150,23] := 840.7844;
   DATA[2150,24] := 2.0;
   DATA[2150,25] := 2.0;
   DATA[2150,26] := 7.874135;
   DATA[2150,27] := 144.1938;
   DATA[2150,28] := 262.0161;
   DATA[2150,29] := 12.03538;
   DATA[2150,30] := 1.723661;
   DATA[2150,31] := 1.291918;
   DATA[2150,32] := 0.7359089;
   DATA[2150,33] := 0.3084265;
   DATA[2150,34] := 2.0;
   DATA[2150,35] := 250.0;
   DATA[2150,36] := 1.69801;
   DATA[2150,37] := 188.8138;
   DATA[2150,38] := 0.000128152;
   DATA[2150,39] := 1.0;
   DATA[2150,40] := 1.0;
   DATA[2151,0] := 2.659578;
   DATA[2151,1] := 863.4037;
   DATA[2151,2] := 2.0;
   DATA[2151,3] := 2.0;
   DATA[2151,4] := 262.3045;
   DATA[2151,5] := 8.392271;
   DATA[2151,6] := 330.6075;
   DATA[2151,7] := 2.463589;
   DATA[2151,8] := 2.0;
   DATA[2151,9] := 2.0;
   DATA[2151,10] := 2.0;
   DATA[2151,11] := 19.65555;
   DATA[2151,12] := 2.209653;
   DATA[2151,13] := 806.524;
   DATA[2151,14] := 1.0;
   DATA[2151,15] := 2.0;
   DATA[2151,16] := 1.0;
   DATA[2151,17] := 1.0;
   DATA[2151,18] := 1.0;
   DATA[2151,19] := 2.0;
   DATA[2151,20] := 148.808;
   DATA[2151,21] := 155.0884;
   DATA[2151,22] := 1.712107;
   DATA[2151,23] := 840.8998;
   DATA[2151,24] := 2.0;
   DATA[2151,25] := 2.0;
   DATA[2151,26] := 7.874135;
   DATA[2151,27] := 144.1938;
   DATA[2151,28] := 261.92;
   DATA[2151,29] := 12.03538;
   DATA[2151,30] := 1.723661;
   DATA[2151,31] := 1.284104;
   DATA[2151,32] := 0.7380853;
   DATA[2151,33] := 0.3084265;
   DATA[2151,34] := 2.0;
   DATA[2151,35] := 250.0;
   DATA[2151,36] := 1.69801;
   DATA[2151,37] := 188.8138;
   DATA[2151,38] := 0.000128152;
   DATA[2151,39] := 1.0;
   DATA[2151,40] := 1.0;
   DATA[2152,0] := 2.633635;
   DATA[2152,1] := 863.4822;
   DATA[2152,2] := 2.0;
   DATA[2152,3] := 2.0;
   DATA[2152,4] := 262.3045;
   DATA[2152,5] := 8.392271;
   DATA[2152,6] := 330.6075;
   DATA[2152,7] := 2.463589;
   DATA[2152,8] := 2.0;
   DATA[2152,9] := 2.0;
   DATA[2152,10] := 2.0;
   DATA[2152,11] := 19.68436;
   DATA[2152,12] := 2.209653;
   DATA[2152,13] := 807.0046;
   DATA[2152,14] := 1.0;
   DATA[2152,15] := 2.0;
   DATA[2152,16] := 1.0;
   DATA[2152,17] := 1.0;
   DATA[2152,18] := 1.0;
   DATA[2152,19] := 2.0;
   DATA[2152,20] := 148.808;
   DATA[2152,21] := 155.0884;
   DATA[2152,22] := 1.712107;
   DATA[2152,23] := 841.2843;
   DATA[2152,24] := 2.0;
   DATA[2152,25] := 2.0;
   DATA[2152,26] := 7.874135;
   DATA[2152,27] := 144.1938;
   DATA[2152,28] := 261.8559;
   DATA[2152,29] := 12.03538;
   DATA[2152,30] := 1.723661;
   DATA[2152,31] := 1.281542;
   DATA[2152,32] := 0.7373172;
   DATA[2152,33] := 0.3084265;
   DATA[2152,34] := 2.0;
   DATA[2152,35] := 250.1602;
   DATA[2152,36] := 1.69801;
   DATA[2152,37] := 188.8138;
   DATA[2152,38] := 0.000128152;
   DATA[2152,39] := 1.0;
   DATA[2152,40] := 1.0;
   DATA[2153,0] := 2.617622;
   DATA[2153,1] := 863.2859;
   DATA[2153,2] := 2.0;
   DATA[2153,3] := 2.0;
   DATA[2153,4] := 262.3045;
   DATA[2153,5] := 8.392271;
   DATA[2153,6] := 330.6075;
   DATA[2153,7] := 2.463589;
   DATA[2153,8] := 2.0;
   DATA[2153,9] := 2.0;
   DATA[2153,10] := 2.0;
   DATA[2153,11] := 19.69396;
   DATA[2153,12] := 2.209653;
   DATA[2153,13] := 807.1649;
   DATA[2153,14] := 1.0;
   DATA[2153,15] := 2.0;
   DATA[2153,16] := 1.0;
   DATA[2153,17] := 1.0;
   DATA[2153,18] := 1.0;
   DATA[2153,19] := 2.0;
   DATA[2153,20] := 148.808;
   DATA[2153,21] := 155.0884;
   DATA[2153,22] := 1.713517;
   DATA[2153,23] := 841.2458;
   DATA[2153,24] := 2.0;
   DATA[2153,25] := 2.0;
   DATA[2153,26] := 7.874135;
   DATA[2153,27] := 144.1938;
   DATA[2153,28] := 261.8559;
   DATA[2153,29] := 12.03538;
   DATA[2153,30] := 1.725327;
   DATA[2153,31] := 1.281542;
   DATA[2153,32] := 0.7360369;
   DATA[2153,33] := 0.3084265;
   DATA[2153,34] := 2.0;
   DATA[2153,35] := 250.2403;
   DATA[2153,36] := 1.69801;
   DATA[2153,37] := 188.9259;
   DATA[2153,38] := 0.000128152;
   DATA[2153,39] := 1.0;
   DATA[2153,40] := 1.0;
   DATA[2154,0] := 2.612497;
   DATA[2154,1] := 863.2466;
   DATA[2154,2] := 2.0;
   DATA[2154,3] := 2.0;
   DATA[2154,4] := 262.3045;
   DATA[2154,5] := 8.392271;
   DATA[2154,6] := 330.6075;
   DATA[2154,7] := 2.463589;
   DATA[2154,8] := 2.0;
   DATA[2154,9] := 2.0;
   DATA[2154,10] := 2.0;
   DATA[2154,11] := 19.69396;
   DATA[2154,12] := 2.209653;
   DATA[2154,13] := 807.285;
   DATA[2154,14] := 1.0;
   DATA[2154,15] := 2.0;
   DATA[2154,16] := 1.0;
   DATA[2154,17] := 1.0;
   DATA[2154,18] := 1.0;
   DATA[2154,19] := 2.0;
   DATA[2154,20] := 148.808;
   DATA[2154,21] := 155.0884;
   DATA[2154,22] := 1.715183;
   DATA[2154,23] := 841.3612;
   DATA[2154,24] := 2.0;
   DATA[2154,25] := 2.0;
   DATA[2154,26] := 7.874135;
   DATA[2154,27] := 144.1938;
   DATA[2154,28] := 261.8559;
   DATA[2154,29] := 12.03538;
   DATA[2154,30] := 1.725327;
   DATA[2154,31] := 1.281542;
   DATA[2154,32] := 0.7360369;
   DATA[2154,33] := 0.3084265;
   DATA[2154,34] := 2.0;
   DATA[2154,35] := 250.2403;
   DATA[2154,36] := 1.842181;
   DATA[2154,37] := 189.022;
   DATA[2154,38] := 0.000128152;
   DATA[2154,39] := 1.0;
   DATA[2154,40] := 1.0;
   DATA[2155,0] := 2.601928;
   DATA[2155,1] := 863.0504;
   DATA[2155,2] := 2.0;
   DATA[2155,3] := 2.0;
   DATA[2155,4] := 262.3045;
   DATA[2155,5] := 8.392271;
   DATA[2155,6] := 330.6075;
   DATA[2155,7] := 2.463589;
   DATA[2155,8] := 2.0;
   DATA[2155,9] := 2.0;
   DATA[2155,10] := 2.0;
   DATA[2155,11] := 19.69396;
   DATA[2155,12] := 2.209653;
   DATA[2155,13] := 807.3651;
   DATA[2155,14] := 1.0;
   DATA[2155,15] := 2.0;
   DATA[2155,16] := 1.0;
   DATA[2155,17] := 1.0;
   DATA[2155,18] := 1.0;
   DATA[2155,19] := 2.0;
   DATA[2155,20] := 148.808;
   DATA[2155,21] := 155.0884;
   DATA[2155,22] := 1.715183;
   DATA[2155,23] := 841.7457;
   DATA[2155,24] := 2.0;
   DATA[2155,25] := 2.0;
   DATA[2155,26] := 7.874135;
   DATA[2155,27] := 144.1938;
   DATA[2155,28] := 261.8559;
   DATA[2155,29] := 12.03538;
   DATA[2155,30] := 1.725327;
   DATA[2155,31] := 1.281542;
   DATA[2155,32] := 0.7352687;
   DATA[2155,33] := 0.3084265;
   DATA[2155,34] := 2.0;
   DATA[2155,35] := 250.2403;
   DATA[2155,36] := 1.842181;
   DATA[2155,37] := 189.022;
   DATA[2155,38] := 0.000128152;
   DATA[2155,39] := 1.0;
   DATA[2155,40] := 1.0;
   DATA[2156,0] := 2.583992;
   DATA[2156,1] := 862.8934;
   DATA[2156,2] := 2.0;
   DATA[2156,3] := 2.0;
   DATA[2156,4] := 262.3045;
   DATA[2156,5] := 8.392271;
   DATA[2156,6] := 330.6075;
   DATA[2156,7] := 2.463589;
   DATA[2156,8] := 2.0;
   DATA[2156,9] := 2.0;
   DATA[2156,10] := 2.0;
   DATA[2156,11] := 19.69396;
   DATA[2156,12] := 2.209653;
   DATA[2156,13] := 807.6055;
   DATA[2156,14] := 1.0;
   DATA[2156,15] := 2.0;
   DATA[2156,16] := 1.0;
   DATA[2156,17] := 1.0;
   DATA[2156,18] := 1.0;
   DATA[2156,19] := 2.0;
   DATA[2156,20] := 148.808;
   DATA[2156,21] := 155.0884;
   DATA[2156,22] := 1.715183;
   DATA[2156,23] := 841.5919;
   DATA[2156,24] := 2.0;
   DATA[2156,25] := 2.0;
   DATA[2156,26] := 7.874135;
   DATA[2156,27] := 144.0144;
   DATA[2156,28] := 261.8559;
   DATA[2156,29] := 12.03538;
   DATA[2156,30] := 1.725327;
   DATA[2156,31] := 1.281542;
   DATA[2156,32] := 0.7352687;
   DATA[2156,33] := 0.3084265;
   DATA[2156,34] := 2.0;
   DATA[2156,35] := 250.2403;
   DATA[2156,36] := 1.842181;
   DATA[2156,37] := 189.022;
   DATA[2156,38] := 0.000128152;
   DATA[2156,39] := 1.0;
   DATA[2156,40] := 1.0;
   DATA[2157,0] := 2.562854;
   DATA[2157,1] := 862.7756;
   DATA[2157,2] := 2.0;
   DATA[2157,3] := 2.0;
   DATA[2157,4] := 262.3045;
   DATA[2157,5] := 8.392271;
   DATA[2157,6] := 330.6075;
   DATA[2157,7] := 2.46141;
   DATA[2157,8] := 2.0;
   DATA[2157,9] := 2.0;
   DATA[2157,10] := 2.0;
   DATA[2157,11] := 19.69396;
   DATA[2157,12] := 2.206963;
   DATA[2157,13] := 807.6055;
   DATA[2157,14] := 1.0;
   DATA[2157,15] := 2.0;
   DATA[2157,16] := 1.0;
   DATA[2157,17] := 1.0;
   DATA[2157,18] := 1.0;
   DATA[2157,19] := 2.0;
   DATA[2157,20] := 148.808;
   DATA[2157,21] := 155.0884;
   DATA[2157,22] := 1.715567;
   DATA[2157,23] := 842.0149;
   DATA[2157,24] := 2.0;
   DATA[2157,25] := 2.0;
   DATA[2157,26] := 7.874135;
   DATA[2157,27] := 144.0144;
   DATA[2157,28] := 261.8559;
   DATA[2157,29] := 12.03538;
   DATA[2157,30] := 1.725327;
   DATA[2157,31] := 1.281542;
   DATA[2157,32] := 0.7352687;
   DATA[2157,33] := 0.3084265;
   DATA[2157,34] := 2.0;
   DATA[2157,35] := 250.2403;
   DATA[2157,36] := 1.842181;
   DATA[2157,37] := 189.022;
   DATA[2157,38] := 0.000128152;
   DATA[2157,39] := 1.0;
   DATA[2157,40] := 1.0;
   DATA[2158,0] := 2.547481;
   DATA[2158,1] := 863.0111;
   DATA[2158,2] := 2.0;
   DATA[2158,3] := 2.0;
   DATA[2158,4] := 262.3045;
   DATA[2158,5] := 8.392271;
   DATA[2158,6] := 330.6075;
   DATA[2158,7] := 2.461026;
   DATA[2158,8] := 2.0;
   DATA[2158,9] := 2.0;
   DATA[2158,10] := 2.0;
   DATA[2158,11] := 19.70357;
   DATA[2158,12] := 2.206963;
   DATA[2158,13] := 808.2062;
   DATA[2158,14] := 1.0;
   DATA[2158,15] := 2.0;
   DATA[2158,16] := 1.0;
   DATA[2158,17] := 1.0;
   DATA[2158,18] := 1.0;
   DATA[2158,19] := 2.0;
   DATA[2158,20] := 148.808;
   DATA[2158,21] := 155.0884;
   DATA[2158,22] := 1.716208;
   DATA[2158,23] := 842.4379;
   DATA[2158,24] := 2.0;
   DATA[2158,25] := 2.0;
   DATA[2158,26] := 7.874135;
   DATA[2158,27] := 144.0144;
   DATA[2158,28] := 261.8559;
   DATA[2158,29] := 12.03538;
   DATA[2158,30] := 1.726352;
   DATA[2158,31] := 1.281542;
   DATA[2158,32] := 0.7352687;
   DATA[2158,33] := 0.3084265;
   DATA[2158,34] := 2.0;
   DATA[2158,35] := 250.2403;
   DATA[2158,36] := 1.730048;
   DATA[2158,37] := 189.022;
   DATA[2158,38] := 0.000128152;
   DATA[2158,39] := 1.0;
   DATA[2158,40] := 1.0;
   DATA[2159,0] := 2.527624;
   DATA[2159,1] := 862.7756;
   DATA[2159,2] := 2.0;
   DATA[2159,3] := 2.0;
   DATA[2159,4] := 262.3045;
   DATA[2159,5] := 8.392271;
   DATA[2159,6] := 330.6075;
   DATA[2159,7] := 2.461026;
   DATA[2159,8] := 2.0;
   DATA[2159,9] := 2.0;
   DATA[2159,10] := 2.0;
   DATA[2159,11] := 19.73878;
   DATA[2159,12] := 2.206963;
   DATA[2159,13] := 808.006;
   DATA[2159,14] := 1.0;
   DATA[2159,15] := 2.0;
   DATA[2159,16] := 1.0;
   DATA[2159,17] := 1.0;
   DATA[2159,18] := 1.0;
   DATA[2159,19] := 2.0;
   DATA[2159,20] := 148.808;
   DATA[2159,21] := 155.0884;
   DATA[2159,22] := 1.716208;
   DATA[2159,23] := 842.707;
   DATA[2159,24] := 2.0;
   DATA[2159,25] := 2.0;
   DATA[2159,26] := 7.874135;
   DATA[2159,27] := 144.0144;
   DATA[2159,28] := 261.8559;
   DATA[2159,29] := 12.03538;
   DATA[2159,30] := 1.726609;
   DATA[2159,31] := 1.270398;
   DATA[2159,32] := 0.7352687;
   DATA[2159,33] := 0.3084265;
   DATA[2159,34] := 2.0;
   DATA[2159,35] := 250.2403;
   DATA[2159,36] := 1.730048;
   DATA[2159,37] := 189.022;
   DATA[2159,38] := 0.000128152;
   DATA[2159,39] := 1.0;
   DATA[2159,40] := 1.0;
   DATA[2160,0] := 2.516414;
   DATA[2160,1] := 862.6578;
   DATA[2160,2] := 2.0;
   DATA[2160,3] := 2.0;
   DATA[2160,4] := 262.3045;
   DATA[2160,5] := 8.392271;
   DATA[2160,6] := 330.6075;
   DATA[2160,7] := 2.463461;
   DATA[2160,8] := 2.0;
   DATA[2160,9] := 2.0;
   DATA[2160,10] := 2.0;
   DATA[2160,11] := 19.73878;
   DATA[2160,12] := 2.206963;
   DATA[2160,13] := 808.6068;
   DATA[2160,14] := 1.0;
   DATA[2160,15] := 2.0;
   DATA[2160,16] := 1.0;
   DATA[2160,17] := 1.0;
   DATA[2160,18] := 1.0;
   DATA[2160,19] := 2.0;
   DATA[2160,20] := 148.808;
   DATA[2160,21] := 155.0884;
   DATA[2160,22] := 1.716208;
   DATA[2160,23] := 842.6301;
   DATA[2160,24] := 2.0;
   DATA[2160,25] := 2.0;
   DATA[2160,26] := 7.874135;
   DATA[2160,27] := 144.0144;
   DATA[2160,28] := 261.8559;
   DATA[2160,29] := 12.03538;
   DATA[2160,30] := 1.726609;
   DATA[2160,31] := 1.270398;
   DATA[2160,32] := 0.7352687;
   DATA[2160,33] := 0.3084265;
   DATA[2160,34] := 2.0;
   DATA[2160,35] := 250.1762;
   DATA[2160,36] := 1.730048;
   DATA[2160,37] := 189.022;
   DATA[2160,38] := 0.000128152;
   DATA[2160,39] := 1.0;
   DATA[2160,40] := 1.0;
   DATA[2161,0] := 2.50008;
   DATA[2161,1] := 862.7756;
   DATA[2161,2] := 2.0;
   DATA[2161,3] := 2.0;
   DATA[2161,4] := 262.3045;
   DATA[2161,5] := 8.392271;
   DATA[2161,6] := 330.6075;
   DATA[2161,7] := 2.463461;
   DATA[2161,8] := 2.0;
   DATA[2161,9] := 2.0;
   DATA[2161,10] := 2.0;
   DATA[2161,11] := 19.69076;
   DATA[2161,12] := 2.206963;
   DATA[2161,13] := 808.3264;
   DATA[2161,14] := 1.0;
   DATA[2161,15] := 2.0;
   DATA[2161,16] := 1.0;
   DATA[2161,17] := 1.0;
   DATA[2161,18] := 1.0;
   DATA[2161,19] := 2.0;
   DATA[2161,20] := 148.808;
   DATA[2161,21] := 155.0884;
   DATA[2161,22] := 1.716208;
   DATA[2161,23] := 843.0915;
   DATA[2161,24] := 2.0;
   DATA[2161,25] := 2.0;
   DATA[2161,26] := 7.873815;
   DATA[2161,27] := 144.0144;
   DATA[2161,28] := 261.8559;
   DATA[2161,29] := 12.03538;
   DATA[2161,30] := 1.72507;
   DATA[2161,31] := 1.272832;
   DATA[2161,32] := 0.7352687;
   DATA[2161,33] := 0.3084265;
   DATA[2161,34] := 2.0;
   DATA[2161,35] := 250.1762;
   DATA[2161,36] := 1.730048;
   DATA[2161,37] := 189.022;
   DATA[2161,38] := 0.000128152;
   DATA[2161,39] := 1.0;
   DATA[2161,40] := 1.0;
   DATA[2162,0] := 2.484707;
   DATA[2162,1] := 862.3831;
   DATA[2162,2] := 2.0;
   DATA[2162,3] := 2.0;
   DATA[2162,4] := 262.3045;
   DATA[2162,5] := 8.392271;
   DATA[2162,6] := 330.6075;
   DATA[2162,7] := 2.463461;
   DATA[2162,8] := 2.0;
   DATA[2162,9] := 2.0;
   DATA[2162,10] := 2.0;
   DATA[2162,11] := 19.69076;
   DATA[2162,12] := 2.206963;
   DATA[2162,13] := 808.4466;
   DATA[2162,14] := 1.0;
   DATA[2162,15] := 2.0;
   DATA[2162,16] := 1.0;
   DATA[2162,17] := 1.0;
   DATA[2162,18] := 1.0;
   DATA[2162,19] := 2.0;
   DATA[2162,20] := 148.808;
   DATA[2162,21] := 155.0884;
   DATA[2162,22] := 1.715952;
   DATA[2162,23] := 842.8223;
   DATA[2162,24] := 2.0;
   DATA[2162,25] := 2.0;
   DATA[2162,26] := 7.873815;
   DATA[2162,27] := 144.0144;
   DATA[2162,28] := 261.8559;
   DATA[2162,29] := 12.03538;
   DATA[2162,30] := 1.72507;
   DATA[2162,31] := 1.28705;
   DATA[2162,32] := 0.7352687;
   DATA[2162,33] := 0.3084265;
   DATA[2162,34] := 2.0;
   DATA[2162,35] := 250.1762;
   DATA[2162,36] := 1.730048;
   DATA[2162,37] := 189.022;
   DATA[2162,38] := 0.000128152;
   DATA[2162,39] := 1.0;
   DATA[2162,40] := 1.0;
   DATA[2163,0] := 2.468052;
   DATA[2163,1] := 862.3831;
   DATA[2163,2] := 2.0;
   DATA[2163,3] := 2.0;
   DATA[2163,4] := 262.3045;
   DATA[2163,5] := 8.392271;
   DATA[2163,6] := 330.6075;
   DATA[2163,7] := 2.463461;
   DATA[2163,8] := 2.0;
   DATA[2163,9] := 2.0;
   DATA[2163,10] := 2.0;
   DATA[2163,11] := 19.69076;
   DATA[2163,12] := 2.206963;
   DATA[2163,13] := 808.3665;
   DATA[2163,14] := 1.0;
   DATA[2163,15] := 2.0;
   DATA[2163,16] := 1.0;
   DATA[2163,17] := 1.0;
   DATA[2163,18] := 1.0;
   DATA[2163,19] := 2.0;
   DATA[2163,20] := 148.808;
   DATA[2163,21] := 155.0884;
   DATA[2163,22] := 1.714798;
   DATA[2163,23] := 842.8992;
   DATA[2163,24] := 2.0;
   DATA[2163,25] := 2.0;
   DATA[2163,26] := 7.873815;
   DATA[2163,27] := 144.0144;
   DATA[2163,28] := 261.8559;
   DATA[2163,29] := 12.03538;
   DATA[2163,30] := 1.72507;
   DATA[2163,31] := 1.29243;
   DATA[2163,32] := 0.7352687;
   DATA[2163,33] := 0.3084265;
   DATA[2163,34] := 2.0;
   DATA[2163,35] := 250.1762;
   DATA[2163,36] := 1.730048;
   DATA[2163,37] := 189.022;
   DATA[2163,38] := 0.000128152;
   DATA[2163,39] := 1.0;
   DATA[2163,40] := 1.0;
   DATA[2164,0] := 2.455562;
   DATA[2164,1] := 862.2653;
   DATA[2164,2] := 2.0;
   DATA[2164,3] := 2.0;
   DATA[2164,4] := 262.3045;
   DATA[2164,5] := 8.392271;
   DATA[2164,6] := 330.6075;
   DATA[2164,7] := 2.463461;
   DATA[2164,8] := 2.0;
   DATA[2164,9] := 2.0;
   DATA[2164,10] := 2.0;
   DATA[2164,11] := 19.65235;
   DATA[2164,12] := 2.209013;
   DATA[2164,13] := 808.5667;
   DATA[2164,14] := 1.0;
   DATA[2164,15] := 2.0;
   DATA[2164,16] := 1.0;
   DATA[2164,17] := 1.0;
   DATA[2164,18] := 1.0;
   DATA[2164,19] := 2.0;
   DATA[2164,20] := 148.808;
   DATA[2164,21] := 155.0884;
   DATA[2164,22] := 1.714798;
   DATA[2164,23] := 843.2068;
   DATA[2164,24] := 2.0;
   DATA[2164,25] := 2.0;
   DATA[2164,26] := 7.873815;
   DATA[2164,27] := 144.0144;
   DATA[2164,28] := 261.8559;
   DATA[2164,29] := 12.03538;
   DATA[2164,30] := 1.72507;
   DATA[2164,31] := 1.29243;
   DATA[2164,32] := 0.7352687;
   DATA[2164,33] := 0.3084265;
   DATA[2164,34] := 2.0;
   DATA[2164,35] := 250.1762;
   DATA[2164,36] := 1.730048;
   DATA[2164,37] := 189.022;
   DATA[2164,38] := 0.000128152;
   DATA[2164,39] := 1.0;
   DATA[2164,40] := 1.0;
   DATA[2165,0] := 2.444992;
   DATA[2165,1] := 862.0691;
   DATA[2165,2] := 2.0;
   DATA[2165,3] := 2.0;
   DATA[2165,4] := 262.3045;
   DATA[2165,5] := 8.392271;
   DATA[2165,6] := 330.6075;
   DATA[2165,7] := 2.463461;
   DATA[2165,8] := 2.0;
   DATA[2165,9] := 2.0;
   DATA[2165,10] := 2.0;
   DATA[2165,11] := 19.65235;
   DATA[2165,12] := 2.209013;
   DATA[2165,13] := 808.6068;
   DATA[2165,14] := 1.0;
   DATA[2165,15] := 2.0;
   DATA[2165,16] := 1.0;
   DATA[2165,17] := 1.0;
   DATA[2165,18] := 1.0;
   DATA[2165,19] := 2.0;
   DATA[2165,20] := 148.808;
   DATA[2165,21] := 155.0884;
   DATA[2165,22] := 1.714798;
   DATA[2165,23] := 843.0146;
   DATA[2165,24] := 2.0;
   DATA[2165,25] := 2.0;
   DATA[2165,26] := 7.873815;
   DATA[2165,27] := 144.0144;
   DATA[2165,28] := 261.8559;
   DATA[2165,29] := 12.03538;
   DATA[2165,30] := 1.72507;
   DATA[2165,31] := 1.29243;
   DATA[2165,32] := 0.7352687;
   DATA[2165,33] := 0.3084265;
   DATA[2165,34] := 2.0;
   DATA[2165,35] := 250.1762;
   DATA[2165,36] := 1.730048;
   DATA[2165,37] := 189.022;
   DATA[2165,38] := 0.000128152;
   DATA[2165,39] := 1.0;
   DATA[2165,40] := 1.0;
   DATA[2166,0] := 2.432181;
   DATA[2166,1] := 862.4224;
   DATA[2166,2] := 2.0;
   DATA[2166,3] := 2.0;
   DATA[2166,4] := 262.3045;
   DATA[2166,5] := 8.392271;
   DATA[2166,6] := 330.6075;
   DATA[2166,7] := 2.463461;
   DATA[2166,8] := 2.0;
   DATA[2166,9] := 2.0;
   DATA[2166,10] := 2.0;
   DATA[2166,11] := 19.72598;
   DATA[2166,12] := 2.209013;
   DATA[2166,13] := 808.6469;
   DATA[2166,14] := 1.0;
   DATA[2166,15] := 2.0;
   DATA[2166,16] := 1.0;
   DATA[2166,17] := 1.0;
   DATA[2166,18] := 1.0;
   DATA[2166,19] := 2.0;
   DATA[2166,20] := 148.808;
   DATA[2166,21] := 155.0884;
   DATA[2166,22] := 1.718002;
   DATA[2166,23] := 842.8223;
   DATA[2166,24] := 2.0;
   DATA[2166,25] := 2.0;
   DATA[2166,26] := 7.873815;
   DATA[2166,27] := 144.0144;
   DATA[2166,28] := 261.8559;
   DATA[2166,29] := 12.03538;
   DATA[2166,30] := 1.72507;
   DATA[2166,31] := 1.29243;
   DATA[2166,32] := 0.7352687;
   DATA[2166,33] := 0.3084265;
   DATA[2166,34] := 2.0;
   DATA[2166,35] := 250.1762;
   DATA[2166,36] := 1.730048;
   DATA[2166,37] := 189.022;
   DATA[2166,38] := 0.000128152;
   DATA[2166,39] := 1.0;
   DATA[2166,40] := 1.0;
   DATA[2167,0] := 2.427057;
   DATA[2167,1] := 862.4616;
   DATA[2167,2] := 2.0;
   DATA[2167,3] := 2.0;
   DATA[2167,4] := 262.3045;
   DATA[2167,5] := 8.392271;
   DATA[2167,6] := 330.6075;
   DATA[2167,7] := 2.463461;
   DATA[2167,8] := 2.0;
   DATA[2167,9] := 2.0;
   DATA[2167,10] := 2.0;
   DATA[2167,11] := 19.72598;
   DATA[2167,12] := 2.209013;
   DATA[2167,13] := 808.4466;
   DATA[2167,14] := 1.0;
   DATA[2167,15] := 2.0;
   DATA[2167,16] := 1.0;
   DATA[2167,17] := 1.0;
   DATA[2167,18] := 1.0;
   DATA[2167,19] := 2.0;
   DATA[2167,20] := 148.808;
   DATA[2167,21] := 155.0884;
   DATA[2167,22] := 1.718002;
   DATA[2167,23] := 843.0915;
   DATA[2167,24] := 2.0;
   DATA[2167,25] := 2.0;
   DATA[2167,26] := 7.873815;
   DATA[2167,27] := 143.9631;
   DATA[2167,28] := 261.8559;
   DATA[2167,29] := 12.03538;
   DATA[2167,30] := 1.72507;
   DATA[2167,31] := 1.302037;
   DATA[2167,32] := 0.7352687;
   DATA[2167,33] := 0.3084265;
   DATA[2167,34] := 2.0;
   DATA[2167,35] := 250.1762;
   DATA[2167,36] := 1.730048;
   DATA[2167,37] := 189.022;
   DATA[2167,38] := 0.000128152;
   DATA[2167,39] := 1.0;
   DATA[2167,40] := 1.0;
   DATA[2168,0] := 2.427057;
   DATA[2168,1] := 862.6578;
   DATA[2168,2] := 2.0;
   DATA[2168,3] := 2.0;
   DATA[2168,4] := 262.3045;
   DATA[2168,5] := 8.392271;
   DATA[2168,6] := 330.6075;
   DATA[2168,7] := 2.461539;
   DATA[2168,8] := 2.0;
   DATA[2168,9] := 2.0;
   DATA[2168,10] := 2.0;
   DATA[2168,11] := 19.72598;
   DATA[2168,12] := 2.207091;
   DATA[2168,13] := 808.9673;
   DATA[2168,14] := 1.0;
   DATA[2168,15] := 2.0;
   DATA[2168,16] := 1.0;
   DATA[2168,17] := 1.0;
   DATA[2168,18] := 1.0;
   DATA[2168,19] := 2.0;
   DATA[2168,20] := 148.808;
   DATA[2168,21] := 155.0884;
   DATA[2168,22] := 1.718002;
   DATA[2168,23] := 842.9761;
   DATA[2168,24] := 2.0;
   DATA[2168,25] := 2.0;
   DATA[2168,26] := 7.873815;
   DATA[2168,27] := 143.758;
   DATA[2168,28] := 261.8559;
   DATA[2168,29] := 12.03538;
   DATA[2168,30] := 1.72507;
   DATA[2168,31] := 1.302421;
   DATA[2168,32] := 0.7352687;
   DATA[2168,33] := 0.3084265;
   DATA[2168,34] := 2.0;
   DATA[2168,35] := 250.1762;
   DATA[2168,36] := 1.730048;
   DATA[2168,37] := 189.022;
   DATA[2168,38] := 0.000128152;
   DATA[2168,39] := 1.0;
   DATA[2168,40] := 1.0;
   DATA[2169,0] := 2.463568;
   DATA[2169,1] := 862.3046;
   DATA[2169,2] := 2.0;
   DATA[2169,3] := 2.0;
   DATA[2169,4] := 262.3045;
   DATA[2169,5] := 8.392271;
   DATA[2169,6] := 330.6075;
   DATA[2169,7] := 2.461539;
   DATA[2169,8] := 2.0;
   DATA[2169,9] := 2.0;
   DATA[2169,10] := 2.0;
   DATA[2169,11] := 19.75799;
   DATA[2169,12] := 2.206707;
   DATA[2169,13] := 808.9272;
   DATA[2169,14] := 1.0;
   DATA[2169,15] := 2.0;
   DATA[2169,16] := 1.0;
   DATA[2169,17] := 1.0;
   DATA[2169,18] := 1.0;
   DATA[2169,19] := 2.0;
   DATA[2169,20] := 148.808;
   DATA[2169,21] := 155.0884;
   DATA[2169,22] := 1.715439;
   DATA[2169,23] := 842.9761;
   DATA[2169,24] := 2.0;
   DATA[2169,25] := 2.0;
   DATA[2169,26] := 7.873815;
   DATA[2169,27] := 143.758;
   DATA[2169,28] := 261.8559;
   DATA[2169,29] := 12.03538;
   DATA[2169,30] := 1.72507;
   DATA[2169,31] := 1.29243;
   DATA[2169,32] := 0.7352687;
   DATA[2169,33] := 0.3084265;
   DATA[2169,34] := 2.0;
   DATA[2169,35] := 250.1762;
   DATA[2169,36] := 1.730048;
   DATA[2169,37] := 189.022;
   DATA[2169,38] := 0.000128152;
   DATA[2169,39] := 1.0;
   DATA[2169,40] := 1.0;
   DATA[2170,0] := 2.501041;
   DATA[2170,1] := 861.9905;
   DATA[2170,2] := 2.0;
   DATA[2170,3] := 2.0;
   DATA[2170,4] := 262.3045;
   DATA[2170,5] := 8.392271;
   DATA[2170,6] := 330.6075;
   DATA[2170,7] := 2.461539;
   DATA[2170,8] := 2.0;
   DATA[2170,9] := 2.0;
   DATA[2170,10] := 2.0;
   DATA[2170,11] := 19.76759;
   DATA[2170,12] := 2.206707;
   DATA[2170,13] := 809.0474;
   DATA[2170,14] := 1.0;
   DATA[2170,15] := 2.0;
   DATA[2170,16] := 1.0;
   DATA[2170,17] := 1.0;
   DATA[2170,18] := 1.0;
   DATA[2170,19] := 2.0;
   DATA[2170,20] := 148.808;
   DATA[2170,21] := 155.0884;
   DATA[2170,22] := 1.715439;
   DATA[2170,23] := 842.8992;
   DATA[2170,24] := 2.0;
   DATA[2170,25] := 2.0;
   DATA[2170,26] := 7.873815;
   DATA[2170,27] := 143.758;
   DATA[2170,28] := 261.8559;
   DATA[2170,29] := 12.03538;
   DATA[2170,30] := 1.725711;
   DATA[2170,31] := 1.283079;
   DATA[2170,32] := 0.7352687;
   DATA[2170,33] := 0.3084265;
   DATA[2170,34] := 2.0;
   DATA[2170,35] := 250.1762;
   DATA[2170,36] := 1.730048;
   DATA[2170,37] := 189.022;
   DATA[2170,38] := 0.000128152;
   DATA[2170,39] := 1.0;
   DATA[2170,40] := 1.0;
   DATA[2171,0] := 2.54684;
   DATA[2171,1] := 862.4224;
   DATA[2171,2] := 2.0;
   DATA[2171,3] := 2.0;
   DATA[2171,4] := 262.3045;
   DATA[2171,5] := 8.392271;
   DATA[2171,6] := 330.6075;
   DATA[2171,7] := 2.461539;
   DATA[2171,8] := 2.0;
   DATA[2171,9] := 2.0;
   DATA[2171,10] := 2.0;
   DATA[2171,11] := 19.7996;
   DATA[2171,12] := 2.208116;
   DATA[2171,13] := 808.8471;
   DATA[2171,14] := 1.0;
   DATA[2171,15] := 2.0;
   DATA[2171,16] := 1.0;
   DATA[2171,17] := 1.0;
   DATA[2171,18] := 1.0;
   DATA[2171,19] := 2.0;
   DATA[2171,20] := 148.808;
   DATA[2171,21] := 155.0884;
   DATA[2171,22] := 1.715439;
   DATA[2171,23] := 842.8992;
   DATA[2171,24] := 2.0;
   DATA[2171,25] := 2.0;
   DATA[2171,26] := 7.873815;
   DATA[2171,27] := 143.758;
   DATA[2171,28] := 261.8559;
   DATA[2171,29] := 12.03538;
   DATA[2171,30] := 1.72789;
   DATA[2171,31] := 1.282567;
   DATA[2171,32] := 0.7352687;
   DATA[2171,33] := 0.3084265;
   DATA[2171,34] := 2.0;
   DATA[2171,35] := 250.3525;
   DATA[2171,36] := 1.730048;
   DATA[2171,37] := 189.022;
   DATA[2171,38] := 0.000128152;
   DATA[2171,39] := 1.0;
   DATA[2171,40] := 1.0;
   DATA[2172,0] := 2.576946;
   DATA[2172,1] := 862.8934;
   DATA[2172,2] := 2.0;
   DATA[2172,3] := 2.0;
   DATA[2172,4] := 262.3686;
   DATA[2172,5] := 8.392271;
   DATA[2172,6] := 330.6075;
   DATA[2172,7] := 2.461539;
   DATA[2172,8] := 2.0;
   DATA[2172,9] := 2.0;
   DATA[2172,10] := 2.0;
   DATA[2172,11] := 19.7996;
   DATA[2172,12] := 2.208116;
   DATA[2172,13] := 809.2076;
   DATA[2172,14] := 1.0;
   DATA[2172,15] := 2.0;
   DATA[2172,16] := 1.0;
   DATA[2172,17] := 1.0;
   DATA[2172,18] := 1.0;
   DATA[2172,19] := 2.0;
   DATA[2172,20] := 148.808;
   DATA[2172,21] := 155.0884;
   DATA[2172,22] := 1.717489;
   DATA[2172,23] := 842.9377;
   DATA[2172,24] := 2.0;
   DATA[2172,25] := 2.0;
   DATA[2172,26] := 7.873815;
   DATA[2172,27] := 143.758;
   DATA[2172,28] := 261.8559;
   DATA[2172,29] := 12.03538;
   DATA[2172,30] := 1.72789;
   DATA[2172,31] := 1.290637;
   DATA[2172,32] := 0.7352687;
   DATA[2172,33] := 0.3084265;
   DATA[2172,34] := 2.0;
   DATA[2172,35] := 250.3525;
   DATA[2172,36] := 1.730048;
   DATA[2172,37] := 189.2784;
   DATA[2172,38] := 0.000128152;
   DATA[2172,39] := 1.0;
   DATA[2172,40] := 1.0;
   DATA[2173,0] := 2.617942;
   DATA[2173,1] := 862.8149;
   DATA[2173,2] := 2.0;
   DATA[2173,3] := 2.0;
   DATA[2173,4] := 262.3686;
   DATA[2173,5] := 8.392271;
   DATA[2173,6] := 330.6075;
   DATA[2173,7] := 2.461539;
   DATA[2173,8] := 2.0;
   DATA[2173,9] := 2.0;
   DATA[2173,10] := 2.0;
   DATA[2173,11] := 19.73878;
   DATA[2173,12] := 2.207347;
   DATA[2173,13] := 808.9673;
   DATA[2173,14] := 1.0;
   DATA[2173,15] := 2.0;
   DATA[2173,16] := 1.0;
   DATA[2173,17] := 1.0;
   DATA[2173,18] := 1.0;
   DATA[2173,19] := 2.0;
   DATA[2173,20] := 148.808;
   DATA[2173,21] := 155.0884;
   DATA[2173,22] := 1.717489;
   DATA[2173,23] := 842.8223;
   DATA[2173,24] := 2.0;
   DATA[2173,25] := 2.0;
   DATA[2173,26] := 7.873815;
   DATA[2173,27] := 143.8605;
   DATA[2173,28] := 261.8559;
   DATA[2173,29] := 12.03538;
   DATA[2173,30] := 1.72789;
   DATA[2173,31] := 1.291405;
   DATA[2173,32] := 0.7352687;
   DATA[2173,33] := 0.3084265;
   DATA[2173,34] := 2.0;
   DATA[2173,35] := 250.3525;
   DATA[2173,36] := 1.730048;
   DATA[2173,37] := 189.2784;
   DATA[2173,38] := 0.000128152;
   DATA[2173,39] := 1.0;
   DATA[2173,40] := 1.0;
   DATA[2174,0] := 2.646767;
   DATA[2174,1] := 862.6578;
   DATA[2174,2] := 2.0;
   DATA[2174,3] := 2.0;
   DATA[2174,4] := 262.3686;
   DATA[2174,5] := 8.392271;
   DATA[2174,6] := 330.6075;
   DATA[2174,7] := 2.461539;
   DATA[2174,8] := 2.0;
   DATA[2174,9] := 2.0;
   DATA[2174,10] := 2.0;
   DATA[2174,11] := 19.72277;
   DATA[2174,12] := 2.206963;
   DATA[2174,13] := 809.0474;
   DATA[2174,14] := 1.0;
   DATA[2174,15] := 2.0;
   DATA[2174,16] := 1.0;
   DATA[2174,17] := 1.0;
   DATA[2174,18] := 1.0;
   DATA[2174,19] := 2.0;
   DATA[2174,20] := 148.808;
   DATA[2174,21] := 155.0884;
   DATA[2174,22] := 1.717489;
   DATA[2174,23] := 842.7454;
   DATA[2174,24] := 2.0;
   DATA[2174,25] := 2.0;
   DATA[2174,26] := 7.873815;
   DATA[2174,27] := 143.9887;
   DATA[2174,28] := 261.8559;
   DATA[2174,29] := 12.03538;
   DATA[2174,30] := 1.731223;
   DATA[2174,31] := 1.286922;
   DATA[2174,32] := 0.7352687;
   DATA[2174,33] := 0.3084265;
   DATA[2174,34] := 2.0;
   DATA[2174,35] := 250.4807;
   DATA[2174,36] := 1.730048;
   DATA[2174,37] := 189.2784;
   DATA[2174,38] := 0.000128152;
   DATA[2174,39] := 1.0;
   DATA[2174,40] := 1.0;
   DATA[2175,0] := 2.660539;
   DATA[2175,1] := 862.8934;
   DATA[2175,2] := 2.0;
   DATA[2175,3] := 2.0;
   DATA[2175,4] := 262.3686;
   DATA[2175,5] := 8.392271;
   DATA[2175,6] := 330.6075;
   DATA[2175,7] := 2.461539;
   DATA[2175,8] := 2.0;
   DATA[2175,9] := 2.0;
   DATA[2175,10] := 2.0;
   DATA[2175,11] := 19.72277;
   DATA[2175,12] := 2.206963;
   DATA[2175,13] := 809.2476;
   DATA[2175,14] := 1.0;
   DATA[2175,15] := 2.0;
   DATA[2175,16] := 1.0;
   DATA[2175,17] := 1.0;
   DATA[2175,18] := 1.0;
   DATA[2175,19] := 2.0;
   DATA[2175,20] := 148.808;
   DATA[2175,21] := 155.0884;
   DATA[2175,22] := 1.717489;
   DATA[2175,23] := 842.8992;
   DATA[2175,24] := 2.0;
   DATA[2175,25] := 2.0;
   DATA[2175,26] := 7.873815;
   DATA[2175,27] := 143.9887;
   DATA[2175,28] := 261.8559;
   DATA[2175,29] := 12.03538;
   DATA[2175,30] := 1.731351;
   DATA[2175,31] := 1.300372;
   DATA[2175,32] := 0.7352687;
   DATA[2175,33] := 0.3074016;
   DATA[2175,34] := 2.0;
   DATA[2175,35] := 250.5608;
   DATA[2175,36] := 1.730048;
   DATA[2175,37] := 189.2784;
   DATA[2175,38] := 0.000128152;
   DATA[2175,39] := 1.0;
   DATA[2175,40] := 1.0;
   DATA[2176,0] := 2.660539;
   DATA[2176,1] := 863.0897;
   DATA[2176,2] := 2.0;
   DATA[2176,3] := 2.0;
   DATA[2176,4] := 262.3686;
   DATA[2176,5] := 8.392271;
   DATA[2176,6] := 330.6075;
   DATA[2176,7] := 2.463204;
   DATA[2176,8] := 2.0;
   DATA[2176,9] := 2.0;
   DATA[2176,10] := 2.0;
   DATA[2176,11] := 19.72277;
   DATA[2176,12] := 2.208756;
   DATA[2176,13] := 809.2476;
   DATA[2176,14] := 1.0;
   DATA[2176,15] := 2.0;
   DATA[2176,16] := 1.0;
   DATA[2176,17] := 1.0;
   DATA[2176,18] := 1.0;
   DATA[2176,19] := 2.0;
   DATA[2176,20] := 148.808;
   DATA[2176,21] := 155.0884;
   DATA[2176,22] := 1.717489;
   DATA[2176,23] := 842.7839;
   DATA[2176,24] := 2.0;
   DATA[2176,25] := 2.0;
   DATA[2176,26] := 7.873815;
   DATA[2176,27] := 143.9887;
   DATA[2176,28] := 261.8559;
   DATA[2176,29] := 12.03538;
   DATA[2176,30] := 1.731351;
   DATA[2176,31] := 1.30985;
   DATA[2176,32] := 0.7352687;
   DATA[2176,33] := 0.306761;
   DATA[2176,34] := 2.0;
   DATA[2176,35] := 250.5608;
   DATA[2176,36] := 1.730048;
   DATA[2176,37] := 189.2784;
   DATA[2176,38] := 0.000128152;
   DATA[2176,39] := 1.0;
   DATA[2176,40] := 1.0;
   DATA[2177,0] := 2.636198;
   DATA[2177,1] := 863.3644;
   DATA[2177,2] := 2.0;
   DATA[2177,3] := 2.0;
   DATA[2177,4] := 262.3686;
   DATA[2177,5] := 8.392271;
   DATA[2177,6] := 330.5563;
   DATA[2177,7] := 2.463204;
   DATA[2177,8] := 2.0;
   DATA[2177,9] := 2.0;
   DATA[2177,10] := 2.0;
   DATA[2177,11] := 19.7868;
   DATA[2177,12] := 2.208756;
   DATA[2177,13] := 809.6082;
   DATA[2177,14] := 1.0;
   DATA[2177,15] := 2.0;
   DATA[2177,16] := 1.0;
   DATA[2177,17] := 1.0;
   DATA[2177,18] := 1.0;
   DATA[2177,19] := 2.0;
   DATA[2177,20] := 148.808;
   DATA[2177,21] := 155.0884;
   DATA[2177,22] := 1.71813;
   DATA[2177,23] := 843.2068;
   DATA[2177,24] := 2.0;
   DATA[2177,25] := 2.0;
   DATA[2177,26] := 7.873815;
   DATA[2177,27] := 143.9887;
   DATA[2177,28] := 261.8559;
   DATA[2177,29] := 12.03538;
   DATA[2177,30] := 1.731351;
   DATA[2177,31] := 1.319329;
   DATA[2177,32] := 0.7352687;
   DATA[2177,33] := 0.306761;
   DATA[2177,34] := 2.0;
   DATA[2177,35] := 250.5608;
   DATA[2177,36] := 1.730048;
   DATA[2177,37] := 189.2784;
   DATA[2177,38] := 0.000128152;
   DATA[2177,39] := 1.0;
   DATA[2177,40] := 1.0;
   DATA[2178,0] := 2.623387;
   DATA[2178,1] := 863.8354;
   DATA[2178,2] := 2.0;
   DATA[2178,3] := 2.0;
   DATA[2178,4] := 262.3686;
   DATA[2178,5] := 8.392271;
   DATA[2178,6] := 330.4281;
   DATA[2178,7] := 2.461923;
   DATA[2178,8] := 2.0;
   DATA[2178,9] := 2.0;
   DATA[2178,10] := 2.0;
   DATA[2178,11] := 19.7868;
   DATA[2178,12] := 2.208756;
   DATA[2178,13] := 809.5681;
   DATA[2178,14] := 1.0;
   DATA[2178,15] := 2.0;
   DATA[2178,16] := 1.0;
   DATA[2178,17] := 1.0;
   DATA[2178,18] := 1.0;
   DATA[2178,19] := 2.0;
   DATA[2178,20] := 148.808;
   DATA[2178,21] := 155.0884;
   DATA[2178,22] := 1.71813;
   DATA[2178,23] := 843.476;
   DATA[2178,24] := 2.0;
   DATA[2178,25] := 2.0;
   DATA[2178,26] := 7.873815;
   DATA[2178,27] := 143.9887;
   DATA[2178,28] := 261.8559;
   DATA[2178,29] := 12.03538;
   DATA[2178,30] := 1.731351;
   DATA[2178,31] := 1.322531;
   DATA[2178,32] := 0.7352687;
   DATA[2178,33] := 0.3084905;
   DATA[2178,34] := 2.0;
   DATA[2178,35] := 250.5608;
   DATA[2178,36] := 1.730048;
   DATA[2178,37] := 189.2784;
   DATA[2178,38] := 0.000128152;
   DATA[2178,39] := 1.0;
   DATA[2178,40] := 1.0;
   DATA[2179,0] := 2.616981;
   DATA[2179,1] := 864.1495;
   DATA[2179,2] := 2.0;
   DATA[2179,3] := 2.0;
   DATA[2179,4] := 262.3686;
   DATA[2179,5] := 8.392271;
   DATA[2179,6] := 330.3256;
   DATA[2179,7] := 2.46141;
   DATA[2179,8] := 2.0;
   DATA[2179,9] := 2.0;
   DATA[2179,10] := 2.0;
   DATA[2179,11] := 19.7868;
   DATA[2179,12] := 2.209269;
   DATA[2179,13] := 809.6482;
   DATA[2179,14] := 1.0;
   DATA[2179,15] := 2.0;
   DATA[2179,16] := 1.0;
   DATA[2179,17] := 1.0;
   DATA[2179,18] := 1.0;
   DATA[2179,19] := 2.0;
   DATA[2179,20] := 148.808;
   DATA[2179,21] := 155.0884;
   DATA[2179,22] := 1.71813;
   DATA[2179,23] := 843.476;
   DATA[2179,24] := 2.0;
   DATA[2179,25] := 2.0;
   DATA[2179,26] := 7.873815;
   DATA[2179,27] := 143.9887;
   DATA[2179,28] := 261.8559;
   DATA[2179,29] := 12.03538;
   DATA[2179,30] := 1.731351;
   DATA[2179,31] := 1.322531;
   DATA[2179,32] := 0.7352687;
   DATA[2179,33] := 0.3084905;
   DATA[2179,34] := 2.0;
   DATA[2179,35] := 250.5608;
   DATA[2179,36] := 1.730048;
   DATA[2179,37] := 189.2784;
   DATA[2179,38] := 0.000128152;
   DATA[2179,39] := 1.0;
   DATA[2179,40] := 1.0;
   DATA[2180,0] := 2.612177;
   DATA[2180,1] := 863.9532;
   DATA[2180,2] := 2.0;
   DATA[2180,3] := 2.0;
   DATA[2180,4] := 262.3686;
   DATA[2180,5] := 8.392271;
   DATA[2180,6] := 330.3256;
   DATA[2180,7] := 2.46141;
   DATA[2180,8] := 2.0;
   DATA[2180,9] := 2.0;
   DATA[2180,10] := 2.0;
   DATA[2180,11] := 19.7868;
   DATA[2180,12] := 2.210037;
   DATA[2180,13] := 810.1288;
   DATA[2180,14] := 1.0;
   DATA[2180,15] := 2.0;
   DATA[2180,16] := 1.0;
   DATA[2180,17] := 1.0;
   DATA[2180,18] := 1.0;
   DATA[2180,19] := 2.0;
   DATA[2180,20] := 148.808;
   DATA[2180,21] := 155.0884;
   DATA[2180,22] := 1.715952;
   DATA[2180,23] := 843.9374;
   DATA[2180,24] := 2.0;
   DATA[2180,25] := 2.0;
   DATA[2180,26] := 7.873815;
   DATA[2180,27] := 143.9887;
   DATA[2180,28] := 262.0161;
   DATA[2180,29] := 12.03538;
   DATA[2180,30] := 1.731351;
   DATA[2180,31] := 1.313693;
   DATA[2180,32] := 0.7352687;
   DATA[2180,33] := 0.3084905;
   DATA[2180,34] := 2.0;
   DATA[2180,35] := 250.5608;
   DATA[2180,36] := 1.730048;
   DATA[2180,37] := 189.2784;
   DATA[2180,38] := 0.000128152;
   DATA[2180,39] := 1.0;
   DATA[2180,40] := 1.0;
   DATA[2181,0] := 2.596804;
   DATA[2181,1] := 863.9532;
   DATA[2181,2] := 2.0;
   DATA[2181,3] := 2.0;
   DATA[2181,4] := 262.3686;
   DATA[2181,5] := 8.392271;
   DATA[2181,6] := 330.3256;
   DATA[2181,7] := 2.46077;
   DATA[2181,8] := 2.0;
   DATA[2181,9] := 2.0;
   DATA[2181,10] := 2.0;
   DATA[2181,11] := 19.7868;
   DATA[2181,12] := 2.210037;
   DATA[2181,13] := 810.0087;
   DATA[2181,14] := 1.0;
   DATA[2181,15] := 2.0;
   DATA[2181,16] := 1.0;
   DATA[2181,17] := 1.0;
   DATA[2181,18] := 1.0;
   DATA[2181,19] := 2.0;
   DATA[2181,20] := 148.808;
   DATA[2181,21] := 155.0884;
   DATA[2181,22] := 1.714158;
   DATA[2181,23] := 843.7836;
   DATA[2181,24] := 2.0;
   DATA[2181,25] := 2.0;
   DATA[2181,26] := 7.873815;
   DATA[2181,27] := 143.9887;
   DATA[2181,28] := 262.0161;
   DATA[2181,29] := 12.03538;
   DATA[2181,30] := 1.731351;
   DATA[2181,31] := 1.302933;
   DATA[2181,32] := 0.7352687;
   DATA[2181,33] := 0.3084905;
   DATA[2181,34] := 2.0;
   DATA[2181,35] := 250.4646;
   DATA[2181,36] := 1.730048;
   DATA[2181,37] := 189.2784;
   DATA[2181,38] := 0.000128152;
   DATA[2181,39] := 1.0;
   DATA[2181,40] := 1.0;
   DATA[2182,0] := 2.576946;
   DATA[2182,1] := 864.1887;
   DATA[2182,2] := 2.0;
   DATA[2182,3] := 2.0;
   DATA[2182,4] := 262.3686;
   DATA[2182,5] := 8.392271;
   DATA[2182,6] := 330.3256;
   DATA[2182,7] := 2.46077;
   DATA[2182,8] := 2.0;
   DATA[2182,9] := 2.0;
   DATA[2182,10] := 2.0;
   DATA[2182,11] := 19.74838;
   DATA[2182,12] := 2.210037;
   DATA[2182,13] := 810.249;
   DATA[2182,14] := 1.0;
   DATA[2182,15] := 2.0;
   DATA[2182,16] := 1.0;
   DATA[2182,17] := 1.0;
   DATA[2182,18] := 1.0;
   DATA[2182,19] := 2.0;
   DATA[2182,20] := 148.808;
   DATA[2182,21] := 155.0884;
   DATA[2182,22] := 1.713261;
   DATA[2182,23] := 844.1297;
   DATA[2182,24] := 2.0;
   DATA[2182,25] := 2.0;
   DATA[2182,26] := 7.873815;
   DATA[2182,27] := 143.9887;
   DATA[2182,28] := 262.0161;
   DATA[2182,29] := 12.03538;
   DATA[2182,30] := 1.731351;
   DATA[2182,31] := 1.29243;
   DATA[2182,32] := 0.7352687;
   DATA[2182,33] := 0.3084905;
   DATA[2182,34] := 2.0;
   DATA[2182,35] := 250.4326;
   DATA[2182,36] := 1.649953;
   DATA[2182,37] := 189.2784;
   DATA[2182,38] := 0.000128152;
   DATA[2182,39] := 1.0;
   DATA[2182,40] := 1.0;
   DATA[2183,0] := 2.576946;
   DATA[2183,1] := 864.1887;
   DATA[2183,2] := 2.0;
   DATA[2183,3] := 2.0;
   DATA[2183,4] := 262.3686;
   DATA[2183,5] := 8.392271;
   DATA[2183,6] := 330.3256;
   DATA[2183,7] := 2.46077;
   DATA[2183,8] := 2.0;
   DATA[2183,9] := 2.0;
   DATA[2183,10] := 2.0;
   DATA[2183,11] := 19.74838;
   DATA[2183,12] := 2.210037;
   DATA[2183,13] := 810.249;
   DATA[2183,14] := 1.0;
   DATA[2183,15] := 2.0;
   DATA[2183,16] := 1.0;
   DATA[2183,17] := 1.0;
   DATA[2183,18] := 1.0;
   DATA[2183,19] := 2.0;
   DATA[2183,20] := 148.808;
   DATA[2183,21] := 155.0884;
   DATA[2183,22] := 1.713261;
   DATA[2183,23] := 844.1297;
   DATA[2183,24] := 2.0;
   DATA[2183,25] := 2.0;
   DATA[2183,26] := 7.873815;
   DATA[2183,27] := 143.9887;
   DATA[2183,28] := 262.0161;
   DATA[2183,29] := 12.03538;
   DATA[2183,30] := 1.731351;
   DATA[2183,31] := 1.29243;
   DATA[2183,32] := 0.7352687;
   DATA[2183,33] := 0.3084905;
   DATA[2183,34] := 2.0;
   DATA[2183,35] := 250.4326;
   DATA[2183,36] := 1.649953;
   DATA[2183,37] := 189.2784;
   DATA[2183,38] := 0.000128152;
   DATA[2183,39] := 1.0;
   DATA[2183,40] := 1.0;
   DATA[2184,0] := 2.561253;
   DATA[2184,1] := 864.4243;
   DATA[2184,2] := 2.0;
   DATA[2184,3] := 2.0;
   DATA[2184,4] := 262.3686;
   DATA[2184,5] := 8.392271;
   DATA[2184,6] := 330.3256;
   DATA[2184,7] := 2.460641;
   DATA[2184,8] := 2.0;
   DATA[2184,9] := 2.0;
   DATA[2184,10] := 2.0;
   DATA[2184,11] := 19.72277;
   DATA[2184,12] := 2.208628;
   DATA[2184,13] := 810.5294;
   DATA[2184,14] := 1.0;
   DATA[2184,15] := 2.0;
   DATA[2184,16] := 1.0;
   DATA[2184,17] := 1.0;
   DATA[2184,18] := 1.0;
   DATA[2184,19] := 2.0;
   DATA[2184,20] := 148.808;
   DATA[2184,21] := 155.1397;
   DATA[2184,22] := 1.712748;
   DATA[2184,23] := 844.4758;
   DATA[2184,24] := 2.0;
   DATA[2184,25] := 2.0;
   DATA[2184,26] := 7.873815;
   DATA[2184,27] := 143.9887;
   DATA[2184,28] := 262.0161;
   DATA[2184,29] := 12.03538;
   DATA[2184,30] := 1.731351;
   DATA[2184,31] := 1.280261;
   DATA[2184,32] := 0.7352687;
   DATA[2184,33] := 0.3084905;
   DATA[2184,34] := 2.0;
   DATA[2184,35] := 250.2563;
   DATA[2184,36] := 1.649953;
   DATA[2184,37] := 189.2784;
   DATA[2184,38] := 0.000128152;
   DATA[2184,39] := 1.0;
   DATA[2184,40] := 1.0;
   DATA[2185,0] := 2.541716;
   DATA[2185,1] := 864.8168;
   DATA[2185,2] := 2.0;
   DATA[2185,3] := 2.0;
   DATA[2185,4] := 262.3686;
   DATA[2185,5] := 8.392271;
   DATA[2185,6] := 330.5563;
   DATA[2185,7] := 2.457438;
   DATA[2185,8] := 2.0;
   DATA[2185,9] := 2.0;
   DATA[2185,10] := 2.0;
   DATA[2185,11] := 19.65875;
   DATA[2185,12] := 2.208244;
   DATA[2185,13] := 810.3291;
   DATA[2185,14] := 1.0;
   DATA[2185,15] := 2.0;
   DATA[2185,16] := 1.0;
   DATA[2185,17] := 1.0;
   DATA[2185,18] := 1.0;
   DATA[2185,19] := 2.0;
   DATA[2185,20] := 148.808;
   DATA[2185,21] := 155.1397;
   DATA[2185,22] := 1.712748;
   DATA[2185,23] := 844.322;
   DATA[2185,24] := 2.0;
   DATA[2185,25] := 2.0;
   DATA[2185,26] := 7.873815;
   DATA[2185,27] := 143.9887;
   DATA[2185,28] := 262.0161;
   DATA[2185,29] := 12.03538;
   DATA[2185,30] := 1.731351;
   DATA[2185,31] := 1.273473;
   DATA[2185,32] := 0.7352687;
   DATA[2185,33] := 0.3084905;
   DATA[2185,34] := 2.0;
   DATA[2185,35] := 250.2563;
   DATA[2185,36] := 1.649953;
   DATA[2185,37] := 189.2464;
   DATA[2185,38] := 0.000128152;
   DATA[2185,39] := 1.0;
   DATA[2185,40] := 1.0;
   DATA[2186,0] := 2.532108;
   DATA[2186,1] := 864.9738;
   DATA[2186,2] := 2.0;
   DATA[2186,3] := 2.0;
   DATA[2186,4] := 262.3686;
   DATA[2186,5] := 8.392271;
   DATA[2186,6] := 330.5819;
   DATA[2186,7] := 2.457438;
   DATA[2186,8] := 2.0;
   DATA[2186,9] := 2.0;
   DATA[2186,10] := 2.0;
   DATA[2186,11] := 19.64594;
   DATA[2186,12] := 2.208244;
   DATA[2186,13] := 810.3291;
   DATA[2186,14] := 1.0;
   DATA[2186,15] := 2.0;
   DATA[2186,16] := 1.0;
   DATA[2186,17] := 1.0;
   DATA[2186,18] := 1.0;
   DATA[2186,19] := 2.0;
   DATA[2186,20] := 148.808;
   DATA[2186,21] := 155.1397;
   DATA[2186,22] := 1.712748;
   DATA[2186,23] := 844.322;
   DATA[2186,24] := 2.0;
   DATA[2186,25] := 2.0;
   DATA[2186,26] := 7.873815;
   DATA[2186,27] := 143.9887;
   DATA[2186,28] := 262.0161;
   DATA[2186,29] := 12.03538;
   DATA[2186,30] := 1.72789;
   DATA[2186,31] := 1.282567;
   DATA[2186,32] := 0.7352687;
   DATA[2186,33] := 0.3084905;
   DATA[2186,34] := 2.0;
   DATA[2186,35] := 250.2563;
   DATA[2186,36] := 1.649953;
   DATA[2186,37] := 189.1182;
   DATA[2186,38] := 0.000128152;
   DATA[2186,39] := 1.0;
   DATA[2186,40] := 1.0;
   DATA[2187,0] := 2.51161;
   DATA[2187,1] := 864.7775;
   DATA[2187,2] := 2.0;
   DATA[2187,3] := 2.0;
   DATA[2187,4] := 262.3686;
   DATA[2187,5] := 8.392271;
   DATA[2187,6] := 330.5819;
   DATA[2187,7] := 2.457438;
   DATA[2187,8] := 2.0;
   DATA[2187,9] := 2.0;
   DATA[2187,10] := 2.0;
   DATA[2187,11] := 19.66835;
   DATA[2187,12] := 2.208884;
   DATA[2187,13] := 810.4493;
   DATA[2187,14] := 1.0;
   DATA[2187,15] := 2.0;
   DATA[2187,16] := 1.0;
   DATA[2187,17] := 1.0;
   DATA[2187,18] := 1.0;
   DATA[2187,19] := 2.0;
   DATA[2187,20] := 148.808;
   DATA[2187,21] := 155.1397;
   DATA[2187,22] := 1.713261;
   DATA[2187,23] := 845.0141;
   DATA[2187,24] := 2.0;
   DATA[2187,25] := 2.0;
   DATA[2187,26] := 7.873815;
   DATA[2187,27] := 143.9887;
   DATA[2187,28] := 262.0161;
   DATA[2187,29] := 12.03538;
   DATA[2187,30] := 1.727634;
   DATA[2187,31] := 1.291149;
   DATA[2187,32] := 0.7352687;
   DATA[2187,33] := 0.3084905;
   DATA[2187,34] := 2.0;
   DATA[2187,35] := 250.2563;
   DATA[2187,36] := 1.649953;
   DATA[2187,37] := 189.1182;
   DATA[2187,38] := 0.000128152;
   DATA[2187,39] := 1.0;
   DATA[2187,40] := 1.0;
   DATA[2188,0] := 2.501041;
   DATA[2188,1] := 864.9345;
   DATA[2188,2] := 2.0;
   DATA[2188,3] := 2.0;
   DATA[2188,4] := 262.3686;
   DATA[2188,5] := 8.392271;
   DATA[2188,6] := 330.5819;
   DATA[2188,7] := 2.458719;
   DATA[2188,8] := 2.0;
   DATA[2188,9] := 2.0;
   DATA[2188,10] := 2.0;
   DATA[2188,11] := 19.70357;
   DATA[2188,12] := 2.209397;
   DATA[2188,13] := 810.249;
   DATA[2188,14] := 1.0;
   DATA[2188,15] := 2.0;
   DATA[2188,16] := 1.0;
   DATA[2188,17] := 1.0;
   DATA[2188,18] := 1.0;
   DATA[2188,19] := 2.0;
   DATA[2188,20] := 148.808;
   DATA[2188,21] := 155.1397;
   DATA[2188,22] := 1.715439;
   DATA[2188,23] := 845.0526;
   DATA[2188,24] := 2.0;
   DATA[2188,25] := 2.0;
   DATA[2188,26] := 7.873815;
   DATA[2188,27] := 143.9887;
   DATA[2188,28] := 261.8559;
   DATA[2188,29] := 12.03538;
   DATA[2188,30] := 1.725327;
   DATA[2188,31] := 1.292174;
   DATA[2188,32] := 0.7352687;
   DATA[2188,33] := 0.3084905;
   DATA[2188,34] := 2.0;
   DATA[2188,35] := 250.2563;
   DATA[2188,36] := 1.649953;
   DATA[2188,37] := 189.1182;
   DATA[2188,38] := 0.000128152;
   DATA[2188,39] := 1.0;
   DATA[2188,40] := 1.0;
   DATA[2189,0] := 2.479582;
   DATA[2189,1] := 864.7775;
   DATA[2189,2] := 2.0;
   DATA[2189,3] := 2.0;
   DATA[2189,4] := 262.3686;
   DATA[2189,5] := 8.392271;
   DATA[2189,6] := 330.5819;
   DATA[2189,7] := 2.458719;
   DATA[2189,8] := 2.0;
   DATA[2189,9] := 2.0;
   DATA[2189,10] := 2.0;
   DATA[2189,11] := 19.74198;
   DATA[2189,12] := 2.209397;
   DATA[2189,13] := 810.249;
   DATA[2189,14] := 1.0;
   DATA[2189,15] := 2.0;
   DATA[2189,16] := 1.0;
   DATA[2189,17] := 1.0;
   DATA[2189,18] := 1.0;
   DATA[2189,19] := 2.0;
   DATA[2189,20] := 148.808;
   DATA[2189,21] := 155.1397;
   DATA[2189,22] := 1.715439;
   DATA[2189,23] := 845.2833;
   DATA[2189,24] := 2.0;
   DATA[2189,25] := 2.0;
   DATA[2189,26] := 7.873815;
   DATA[2189,27] := 143.9887;
   DATA[2189,28] := 261.8559;
   DATA[2189,29] := 12.03538;
   DATA[2189,30] := 1.725327;
   DATA[2189,31] := 1.286794;
   DATA[2189,32] := 0.7352687;
   DATA[2189,33] := 0.3080421;
   DATA[2189,34] := 2.0;
   DATA[2189,35] := 250.2563;
   DATA[2189,36] := 1.649953;
   DATA[2189,37] := 189.0541;
   DATA[2189,38] := 0.000128152;
   DATA[2189,39] := 1.0;
   DATA[2189,40] := 1.0;
   DATA[2190,0] := 2.469654;
   DATA[2190,1] := 864.9345;
   DATA[2190,2] := 2.0;
   DATA[2190,3] := 2.0;
   DATA[2190,4] := 262.3686;
   DATA[2190,5] := 8.392271;
   DATA[2190,6] := 330.5819;
   DATA[2190,7] := 2.458719;
   DATA[2190,8] := 2.0;
   DATA[2190,9] := 2.0;
   DATA[2190,10] := 2.0;
   DATA[2190,11] := 19.74198;
   DATA[2190,12] := 2.209397;
   DATA[2190,13] := 810.6095;
   DATA[2190,14] := 1.0;
   DATA[2190,15] := 2.0;
   DATA[2190,16] := 1.0;
   DATA[2190,17] := 1.0;
   DATA[2190,18] := 1.0;
   DATA[2190,19] := 2.0;
   DATA[2190,20] := 148.808;
   DATA[2190,21] := 155.1397;
   DATA[2190,22] := 1.715439;
   DATA[2190,23] := 845.514;
   DATA[2190,24] := 2.0;
   DATA[2190,25] := 2.0;
   DATA[2190,26] := 7.873815;
   DATA[2190,27] := 143.9887;
   DATA[2190,28] := 261.8559;
   DATA[2190,29] := 12.03538;
   DATA[2190,30] := 1.725327;
   DATA[2190,31] := 1.279749;
   DATA[2190,32] := 0.7352687;
   DATA[2190,33] := 0.3065048;
   DATA[2190,34] := 2.0;
   DATA[2190,35] := 250.2563;
   DATA[2190,36] := 1.69801;
   DATA[2190,37] := 189.0541;
   DATA[2190,38] := 0.000128152;
   DATA[2190,39] := 1.0;
   DATA[2190,40] := 1.0;
   DATA[2191,0] := 2.452999;
   DATA[2191,1] := 864.8168;
   DATA[2191,2] := 2.0;
   DATA[2191,3] := 2.0;
   DATA[2191,4] := 262.3686;
   DATA[2191,5] := 8.392271;
   DATA[2191,6] := 330.5563;
   DATA[2191,7] := 2.456925;
   DATA[2191,8] := 2.0;
   DATA[2191,9] := 2.0;
   DATA[2191,10] := 2.0;
   DATA[2191,11] := 19.74198;
   DATA[2191,12] := 2.209397;
   DATA[2191,13] := 810.6095;
   DATA[2191,14] := 1.0;
   DATA[2191,15] := 2.0;
   DATA[2191,16] := 1.0;
   DATA[2191,17] := 1.0;
   DATA[2191,18] := 1.0;
   DATA[2191,19] := 2.0;
   DATA[2191,20] := 148.808;
   DATA[2191,21] := 155.1397;
   DATA[2191,22] := 1.715439;
   DATA[2191,23] := 845.4755;
   DATA[2191,24] := 2.0;
   DATA[2191,25] := 2.0;
   DATA[2191,26] := 7.873815;
   DATA[2191,27] := 143.9887;
   DATA[2191,28] := 261.8559;
   DATA[2191,29] := 12.30454;
   DATA[2191,30] := 1.726993;
   DATA[2191,31] := 1.274625;
   DATA[2191,32] := 0.7352687;
   DATA[2191,33] := 0.3065048;
   DATA[2191,34] := 2.0;
   DATA[2191,35] := 250.2563;
   DATA[2191,36] := 1.69801;
   DATA[2191,37] := 189.0541;
   DATA[2191,38] := 0.000128152;
   DATA[2191,39] := 1.0;
   DATA[2191,40] := 1.0;
   DATA[2192,0] := 2.443391;
   DATA[2192,1] := 865.013;
   DATA[2192,2] := 2.0;
   DATA[2192,3] := 2.0;
   DATA[2192,4] := 262.3686;
   DATA[2192,5] := 8.392271;
   DATA[2192,6] := 330.4281;
   DATA[2192,7] := 2.456412;
   DATA[2192,8] := 2.0;
   DATA[2192,9] := 2.0;
   DATA[2192,10] := 2.0;
   DATA[2192,11] := 19.72598;
   DATA[2192,12] := 2.209397;
   DATA[2192,13] := 810.7296;
   DATA[2192,14] := 1.0;
   DATA[2192,15] := 2.0;
   DATA[2192,16] := 1.0;
   DATA[2192,17] := 1.0;
   DATA[2192,18] := 1.0;
   DATA[2192,19] := 2.0;
   DATA[2192,20] := 148.808;
   DATA[2192,21] := 154.909;
   DATA[2192,22] := 1.716849;
   DATA[2192,23] := 845.6293;
   DATA[2192,24] := 2.0;
   DATA[2192,25] := 2.0;
   DATA[2192,26] := 7.873815;
   DATA[2192,27] := 143.9887;
   DATA[2192,28] := 261.8559;
   DATA[2192,29] := 12.30454;
   DATA[2192,30] := 1.726993;
   DATA[2192,31] := 1.26694;
   DATA[2192,32] := 0.7352687;
   DATA[2192,33] := 0.3081703;
   DATA[2192,34] := 2.0;
   DATA[2192,35] := 250.2563;
   DATA[2192,36] := 1.69801;
   DATA[2192,37] := 189.0541;
   DATA[2192,38] := 0.000128152;
   DATA[2192,39] := 1.0;
   DATA[2192,40] := 1.0;
   DATA[2193,0] := 2.427057;
   DATA[2193,1] := 864.3457;
   DATA[2193,2] := 2.0;
   DATA[2193,3] := 2.0;
   DATA[2193,4] := 262.3686;
   DATA[2193,5] := 8.392271;
   DATA[2193,6] := 330.4281;
   DATA[2193,7] := 2.455772;
   DATA[2193,8] := 2.0;
   DATA[2193,9] := 2.0;
   DATA[2193,10] := 2.0;
   DATA[2193,11] := 19.72598;
   DATA[2193,12] := 2.209397;
   DATA[2193,13] := 810.3691;
   DATA[2193,14] := 1.0;
   DATA[2193,15] := 2.0;
   DATA[2193,16] := 1.0;
   DATA[2193,17] := 1.0;
   DATA[2193,18] := 1.0;
   DATA[2193,19] := 2.0;
   DATA[2193,20] := 148.808;
   DATA[2193,21] := 154.909;
   DATA[2193,22] := 1.716849;
   DATA[2193,23] := 845.514;
   DATA[2193,24] := 2.0;
   DATA[2193,25] := 2.0;
   DATA[2193,26] := 7.873815;
   DATA[2193,27] := 143.9887;
   DATA[2193,28] := 261.8559;
   DATA[2193,29] := 12.30454;
   DATA[2193,30] := 1.728916;
   DATA[2193,31] := 1.272064;
   DATA[2193,32] := 0.7352687;
   DATA[2193,33] := 0.3084265;
   DATA[2193,34] := 2.0;
   DATA[2193,35] := 250.2563;
   DATA[2193,36] := 1.69801;
   DATA[2193,37] := 189.1342;
   DATA[2193,38] := 0.000128152;
   DATA[2193,39] := 1.0;
   DATA[2193,40] := 1.0;
   DATA[2194,0] := 2.427057;
   DATA[2194,1] := 864.4635;
   DATA[2194,2] := 2.0;
   DATA[2194,3] := 2.0;
   DATA[2194,4] := 262.3686;
   DATA[2194,5] := 8.394514;
   DATA[2194,6] := 330.4281;
   DATA[2194,7] := 2.455772;
   DATA[2194,8] := 2.0;
   DATA[2194,9] := 2.0;
   DATA[2194,10] := 2.0;
   DATA[2194,11] := 19.77399;
   DATA[2194,12] := 2.209397;
   DATA[2194,13] := 810.6095;
   DATA[2194,14] := 1.0;
   DATA[2194,15] := 2.0;
   DATA[2194,16] := 1.0;
   DATA[2194,17] := 1.0;
   DATA[2194,18] := 1.0;
   DATA[2194,19] := 2.0;
   DATA[2194,20] := 148.808;
   DATA[2194,21] := 154.909;
   DATA[2194,22] := 1.717489;
   DATA[2194,23] := 845.7062;
   DATA[2194,24] := 2.0;
   DATA[2194,25] := 2.0;
   DATA[2194,26] := 7.873815;
   DATA[2194,27] := 143.9887;
   DATA[2194,28] := 261.8559;
   DATA[2194,29] := 12.30454;
   DATA[2194,30] := 1.728916;
   DATA[2194,31] := 1.280646;
   DATA[2194,32] := 0.7352687;
   DATA[2194,33] := 0.3084265;
   DATA[2194,34] := 2.0;
   DATA[2194,35] := 250.3845;
   DATA[2194,36] := 1.69801;
   DATA[2194,37] := 189.2143;
   DATA[2194,38] := 0.000128152;
   DATA[2194,39] := 1.0;
   DATA[2194,40] := 1.0;
   DATA[2195,0] := 2.427057;
   DATA[2195,1] := 864.6205;
   DATA[2195,2] := 2.0;
   DATA[2195,3] := 2.0;
   DATA[2195,4] := 262.3686;
   DATA[2195,5] := 8.394835;
   DATA[2195,6] := 330.4281;
   DATA[2195,7] := 2.455772;
   DATA[2195,8] := 2.0;
   DATA[2195,9] := 2.0;
   DATA[2195,10] := 2.0;
   DATA[2195,11] := 19.77399;
   DATA[2195,12] := 2.209013;
   DATA[2195,13] := 810.2089;
   DATA[2195,14] := 1.0;
   DATA[2195,15] := 2.0;
   DATA[2195,16] := 1.0;
   DATA[2195,17] := 1.0;
   DATA[2195,18] := 1.0;
   DATA[2195,19] := 2.0;
   DATA[2195,20] := 148.808;
   DATA[2195,21] := 154.909;
   DATA[2195,22] := 1.717489;
   DATA[2195,23] := 845.4371;
   DATA[2195,24] := 2.0;
   DATA[2195,25] := 2.0;
   DATA[2195,26] := 7.873815;
   DATA[2195,27] := 143.9887;
   DATA[2195,28] := 261.8559;
   DATA[2195,29] := 12.30454;
   DATA[2195,30] := 1.728916;
   DATA[2195,31] := 1.291149;
   DATA[2195,32] := 0.7352687;
   DATA[2195,33] := 0.3072735;
   DATA[2195,34] := 2.0;
   DATA[2195,35] := 250.3845;
   DATA[2195,36] := 1.69801;
   DATA[2195,37] := 189.2143;
   DATA[2195,38] := 0.000128152;
   DATA[2195,39] := 1.0;
   DATA[2195,40] := 1.0;
   DATA[2196,0] := 2.460686;
   DATA[2196,1] := 864.4635;
   DATA[2196,2] := 2.0;
   DATA[2196,3] := 2.0;
   DATA[2196,4] := 262.3686;
   DATA[2196,5] := 8.394835;
   DATA[2196,6] := 330.4281;
   DATA[2196,7] := 2.455772;
   DATA[2196,8] := 2.0;
   DATA[2196,9] := 2.0;
   DATA[2196,10] := 2.0;
   DATA[2196,11] := 19.73878;
   DATA[2196,12] := 2.209013;
   DATA[2196,13] := 810.249;
   DATA[2196,14] := 1.0;
   DATA[2196,15] := 2.0;
   DATA[2196,16] := 1.0;
   DATA[2196,17] := 1.0;
   DATA[2196,18] := 1.0;
   DATA[2196,19] := 2.0;
   DATA[2196,20] := 148.808;
   DATA[2196,21] := 154.909;
   DATA[2196,22] := 1.717489;
   DATA[2196,23] := 845.514;
   DATA[2196,24] := 2.0;
   DATA[2196,25] := 2.0;
   DATA[2196,26] := 7.873815;
   DATA[2196,27] := 143.9887;
   DATA[2196,28] := 261.8559;
   DATA[2196,29] := 12.03538;
   DATA[2196,30] := 1.728916;
   DATA[2196,31] := 1.291533;
   DATA[2196,32] := 0.7352687;
   DATA[2196,33] := 0.3069532;
   DATA[2196,34] := 2.0;
   DATA[2196,35] := 250.3845;
   DATA[2196,36] := 1.69801;
   DATA[2196,37] := 189.2143;
   DATA[2196,38] := 0.000128152;
   DATA[2196,39] := 1.0;
   DATA[2196,40] := 1.0;
   DATA[2197,0] := 2.510649;
   DATA[2197,1] := 864.542;
   DATA[2197,2] := 2.0;
   DATA[2197,3] := 2.0;
   DATA[2197,4] := 262.3686;
   DATA[2197,5] := 8.394835;
   DATA[2197,6] := 330.6844;
   DATA[2197,7] := 2.455772;
   DATA[2197,8] := 2.0;
   DATA[2197,9] := 2.0;
   DATA[2197,10] := 2.0;
   DATA[2197,11] := 19.67476;
   DATA[2197,12] := 2.209013;
   DATA[2197,13] := 810.6095;
   DATA[2197,14] := 1.0;
   DATA[2197,15] := 2.0;
   DATA[2197,16] := 1.0;
   DATA[2197,17] := 1.0;
   DATA[2197,18] := 1.0;
   DATA[2197,19] := 2.0;
   DATA[2197,20] := 148.808;
   DATA[2197,21] := 154.909;
   DATA[2197,22] := 1.717489;
   DATA[2197,23] := 845.5909;
   DATA[2197,24] := 2.0;
   DATA[2197,25] := 2.0;
   DATA[2197,26] := 7.873815;
   DATA[2197,27] := 143.9887;
   DATA[2197,28] := 261.8559;
   DATA[2197,29] := 12.03538;
   DATA[2197,30] := 1.728916;
   DATA[2197,31] := 1.28103;
   DATA[2197,32] := 0.7352687;
   DATA[2197,33] := 0.3071454;
   DATA[2197,34] := 2.0;
   DATA[2197,35] := 250.3845;
   DATA[2197,36] := 1.69801;
   DATA[2197,37] := 189.2143;
   DATA[2197,38] := 0.000128152;
   DATA[2197,39] := 1.0;
   DATA[2197,40] := 1.0;
   DATA[2198,0] := 2.543958;
   DATA[2198,1] := 864.5812;
   DATA[2198,2] := 2.0;
   DATA[2198,3] := 2.0;
   DATA[2198,4] := 262.3686;
   DATA[2198,5] := 8.394835;
   DATA[2198,6] := 330.6844;
   DATA[2198,7] := 2.455772;
   DATA[2198,8] := 2.0;
   DATA[2198,9] := 2.0;
   DATA[2198,10] := 2.0;
   DATA[2198,11] := 19.65875;
   DATA[2198,12] := 2.209013;
   DATA[2198,13] := 810.5694;
   DATA[2198,14] := 1.0;
   DATA[2198,15] := 2.0;
   DATA[2198,16] := 1.0;
   DATA[2198,17] := 1.0;
   DATA[2198,18] := 1.0;
   DATA[2198,19] := 2.0;
   DATA[2198,20] := 148.808;
   DATA[2198,21] := 154.909;
   DATA[2198,22] := 1.717489;
   DATA[2198,23] := 845.5909;
   DATA[2198,24] := 2.0;
   DATA[2198,25] := 2.0;
   DATA[2198,26] := 7.873815;
   DATA[2198,27] := 143.9887;
   DATA[2198,28] := 261.8559;
   DATA[2198,29] := 12.03538;
   DATA[2198,30] := 1.728147;
   DATA[2198,31] := 1.28103;
   DATA[2198,32] := 0.7352687;
   DATA[2198,33] := 0.3086186;
   DATA[2198,34] := 2.0;
   DATA[2198,35] := 250.3845;
   DATA[2198,36] := 1.69801;
   DATA[2198,37] := 189.2143;
   DATA[2198,38] := 0.000128152;
   DATA[2198,39] := 1.0;
   DATA[2198,40] := 1.0;
   DATA[2199,0] := 2.588797;
   DATA[2199,1] := 864.6205;
   DATA[2199,2] := 2.0;
   DATA[2199,3] := 2.0;
   DATA[2199,4] := 262.3686;
   DATA[2199,5] := 8.394835;
   DATA[2199,6] := 330.6844;
   DATA[2199,7] := 2.455772;
   DATA[2199,8] := 2.0;
   DATA[2199,9] := 2.0;
   DATA[2199,10] := 2.0;
   DATA[2199,11] := 19.65235;
   DATA[2199,12] := 2.209013;
   DATA[2199,13] := 810.8498;
   DATA[2199,14] := 1.0;
   DATA[2199,15] := 2.0;
   DATA[2199,16] := 1.0;
   DATA[2199,17] := 1.0;
   DATA[2199,18] := 1.0;
   DATA[2199,19] := 2.0;
   DATA[2199,20] := 148.808;
   DATA[2199,21] := 154.909;
   DATA[2199,22] := 1.718002;
   DATA[2199,23] := 845.4755;
   DATA[2199,24] := 2.0;
   DATA[2199,25] := 2.0;
   DATA[2199,26] := 7.873815;
   DATA[2199,27] := 143.9887;
   DATA[2199,28] := 261.8559;
   DATA[2199,29] := 12.03538;
   DATA[2199,30] := 1.726609;
   DATA[2199,31] := 1.274625;
   DATA[2199,32] := 0.7352687;
   DATA[2199,33] := 0.3086186;
   DATA[2199,34] := 2.0;
   DATA[2199,35] := 250.3845;
   DATA[2199,36] := 1.69801;
   DATA[2199,37] := 189.0861;
   DATA[2199,38] := 0.000128152;
   DATA[2199,39] := 1.0;
   DATA[2199,40] := 1.0;
   DATA[2200,0] := 2.619223;
   DATA[2200,1] := 864.5812;
   DATA[2200,2] := 2.0;
   DATA[2200,3] := 2.0;
   DATA[2200,4] := 262.3686;
   DATA[2200,5] := 8.396116;
   DATA[2200,6] := 330.3512;
   DATA[2200,7] := 2.455772;
   DATA[2200,8] := 2.0;
   DATA[2200,9] := 2.0;
   DATA[2200,10] := 2.0;
   DATA[2200,11] := 19.70037;
   DATA[2200,12] := 2.209013;
   DATA[2200,13] := 810.7296;
   DATA[2200,14] := 1.0;
   DATA[2200,15] := 2.0;
   DATA[2200,16] := 1.0;
   DATA[2200,17] := 1.0;
   DATA[2200,18] := 1.0;
   DATA[2200,19] := 2.0;
   DATA[2200,20] := 148.808;
   DATA[2200,21] := 154.909;
   DATA[2200,22] := 1.718002;
   DATA[2200,23] := 845.514;
   DATA[2200,24] := 2.0;
   DATA[2200,25] := 2.0;
   DATA[2200,26] := 7.873815;
   DATA[2200,27] := 143.9887;
   DATA[2200,28] := 261.8559;
   DATA[2200,29] := 12.03538;
   DATA[2200,30] := 1.726609;
   DATA[2200,31] := 1.273345;
   DATA[2200,32] := 0.7352687;
   DATA[2200,33] := 0.3077859;
   DATA[2200,34] := 2.0;
   DATA[2200,35] := 250.3845;
   DATA[2200,36] := 1.69801;
   DATA[2200,37] := 189.0861;
   DATA[2200,38] := 0.000128152;
   DATA[2200,39] := 1.0;
   DATA[2200,40] := 1.0;
   DATA[2201,0] := 2.642603;
   DATA[2201,1] := 864.5812;
   DATA[2201,2] := 2.0;
   DATA[2201,3] := 2.0;
   DATA[2201,4] := 262.3686;
   DATA[2201,5] := 8.396116;
   DATA[2201,6] := 330.3512;
   DATA[2201,7] := 2.458206;
   DATA[2201,8] := 2.0;
   DATA[2201,9] := 2.0;
   DATA[2201,10] := 2.0;
   DATA[2201,11] := 19.70997;
   DATA[2201,12] := 2.209013;
   DATA[2201,13] := 811.1702;
   DATA[2201,14] := 1.0;
   DATA[2201,15] := 2.0;
   DATA[2201,16] := 1.0;
   DATA[2201,17] := 1.0;
   DATA[2201,18] := 1.0;
   DATA[2201,19] := 2.0;
   DATA[2201,20] := 148.808;
   DATA[2201,21] := 154.909;
   DATA[2201,22] := 1.718002;
   DATA[2201,23] := 845.4371;
   DATA[2201,24] := 2.0;
   DATA[2201,25] := 2.0;
   DATA[2201,26] := 7.873815;
   DATA[2201,27] := 143.9887;
   DATA[2201,28] := 261.8559;
   DATA[2201,29] := 12.03538;
   DATA[2201,30] := 1.725583;
   DATA[2201,31] := 1.277443;
   DATA[2201,32] := 0.7352687;
   DATA[2201,33] := 0.3069532;
   DATA[2201,34] := 2.0;
   DATA[2201,35] := 250.3845;
   DATA[2201,36] := 1.69801;
   DATA[2201,37] := 189.0861;
   DATA[2201,38] := 0.000128152;
   DATA[2201,39] := 1.0;
   DATA[2201,40] := 1.0;
   DATA[2202,0] := 2.657336;
   DATA[2202,1] := 865.1308;
   DATA[2202,2] := 2.0;
   DATA[2202,3] := 2.0;
   DATA[2202,4] := 262.3686;
   DATA[2202,5] := 8.396116;
   DATA[2202,6] := 330.3512;
   DATA[2202,7] := 2.458206;
   DATA[2202,8] := 2.0;
   DATA[2202,9] := 2.0;
   DATA[2202,10] := 2.0;
   DATA[2202,11] := 19.70997;
   DATA[2202,12] := 2.209013;
   DATA[2202,13] := 811.01;
   DATA[2202,14] := 1.0;
   DATA[2202,15] := 2.0;
   DATA[2202,16] := 1.0;
   DATA[2202,17] := 1.0;
   DATA[2202,18] := 1.0;
   DATA[2202,19] := 2.0;
   DATA[2202,20] := 148.808;
   DATA[2202,21] := 154.909;
   DATA[2202,22] := 1.718002;
   DATA[2202,23] := 845.3217;
   DATA[2202,24] := 2.0;
   DATA[2202,25] := 2.0;
   DATA[2202,26] := 7.873815;
   DATA[2202,27] := 143.9887;
   DATA[2202,28] := 261.8559;
   DATA[2202,29] := 12.03538;
   DATA[2202,30] := 1.725583;
   DATA[2202,31] := 1.271679;
   DATA[2202,32] := 0.7352687;
   DATA[2202,33] := 0.3069532;
   DATA[2202,34] := 2.0;
   DATA[2202,35] := 250.3525;
   DATA[2202,36] := 1.69801;
   DATA[2202,37] := 189.0861;
   DATA[2202,38] := 0.000128152;
   DATA[2202,39] := 1.0;
   DATA[2202,40] := 1.0;
   DATA[2203,0] := 2.657336;
   DATA[2203,1] := 864.4635;
   DATA[2203,2] := 2.0;
   DATA[2203,3] := 2.0;
   DATA[2203,4] := 262.3686;
   DATA[2203,5] := 8.396116;
   DATA[2203,6] := 330.3512;
   DATA[2203,7] := 2.458206;
   DATA[2203,8] := 2.0;
   DATA[2203,9] := 2.0;
   DATA[2203,10] := 2.0;
   DATA[2203,11] := 19.70997;
   DATA[2203,12] := 2.209013;
   DATA[2203,13] := 810.8498;
   DATA[2203,14] := 1.0;
   DATA[2203,15] := 2.0;
   DATA[2203,16] := 1.0;
   DATA[2203,17] := 1.0;
   DATA[2203,18] := 1.0;
   DATA[2203,19] := 2.0;
   DATA[2203,20] := 148.808;
   DATA[2203,21] := 154.909;
   DATA[2203,22] := 1.718002;
   DATA[2203,23] := 845.3217;
   DATA[2203,24] := 2.0;
   DATA[2203,25] := 2.0;
   DATA[2203,26] := 7.873815;
   DATA[2203,27] := 143.9887;
   DATA[2203,28] := 261.8559;
   DATA[2203,29] := 12.03538;
   DATA[2203,30] := 1.724942;
   DATA[2203,31] := 1.27296;
   DATA[2203,32] := 0.7352687;
   DATA[2203,33] := 0.3083624;
   DATA[2203,34] := 2.0;
   DATA[2203,35] := 250.1602;
   DATA[2203,36] := 1.69801;
   DATA[2203,37] := 189.0861;
   DATA[2203,38] := 0.000128152;
   DATA[2203,39] := 1.0;
   DATA[2203,40] := 1.0;
   DATA[2204,0] := 2.638119;
   DATA[2204,1] := 864.4635;
   DATA[2204,2] := 2.0;
   DATA[2204,3] := 2.0;
   DATA[2204,4] := 262.3686;
   DATA[2204,5] := 8.396116;
   DATA[2204,6] := 330.5563;
   DATA[2204,7] := 2.455643;
   DATA[2204,8] := 2.0;
   DATA[2204,9] := 2.0;
   DATA[2204,10] := 2.0;
   DATA[2204,11] := 19.73878;
   DATA[2204,12] := 2.209013;
   DATA[2204,13] := 811.01;
   DATA[2204,14] := 1.0;
   DATA[2204,15] := 2.0;
   DATA[2204,16] := 1.0;
   DATA[2204,17] := 1.0;
   DATA[2204,18] := 1.0;
   DATA[2204,19] := 2.0;
   DATA[2204,20] := 148.808;
   DATA[2204,21] := 154.909;
   DATA[2204,22] := 1.718002;
   DATA[2204,23] := 845.3986;
   DATA[2204,24] := 2.0;
   DATA[2204,25] := 2.0;
   DATA[2204,26] := 7.873815;
   DATA[2204,27] := 143.9887;
   DATA[2204,28] := 261.8559;
   DATA[2204,29] := 12.03538;
   DATA[2204,30] := 1.724942;
   DATA[2204,31] := 1.277956;
   DATA[2204,32] := 0.7352687;
   DATA[2204,33] := 0.3083624;
   DATA[2204,34] := 2.0;
   DATA[2204,35] := 250.1602;
   DATA[2204,36] := 1.69801;
   DATA[2204,37] := 189.0861;
   DATA[2204,38] := 0.000128152;
   DATA[2204,39] := 1.0;
   DATA[2204,40] := 1.0;
   DATA[2205,0] := 2.623707;
   DATA[2205,1] := 864.071;
   DATA[2205,2] := 2.0;
   DATA[2205,3] := 2.0;
   DATA[2205,4] := 262.3686;
   DATA[2205,5] := 8.396116;
   DATA[2205,6] := 330.5563;
   DATA[2205,7] := 2.455643;
   DATA[2205,8] := 2.0;
   DATA[2205,9] := 2.0;
   DATA[2205,10] := 2.0;
   DATA[2205,11] := 19.73878;
   DATA[2205,12] := 2.209013;
   DATA[2205,13] := 811.3705;
   DATA[2205,14] := 1.0;
   DATA[2205,15] := 2.0;
   DATA[2205,16] := 1.0;
   DATA[2205,17] := 1.0;
   DATA[2205,18] := 1.0;
   DATA[2205,19] := 2.0;
   DATA[2205,20] := 148.808;
   DATA[2205,21] := 154.909;
   DATA[2205,22] := 1.718002;
   DATA[2205,23] := 845.3217;
   DATA[2205,24] := 2.0;
   DATA[2205,25] := 2.0;
   DATA[2205,26] := 7.873815;
   DATA[2205,27] := 143.9887;
   DATA[2205,28] := 261.8559;
   DATA[2205,29] := 12.03538;
   DATA[2205,30] := 1.724942;
   DATA[2205,31] := 1.277315;
   DATA[2205,32] := 0.7352687;
   DATA[2205,33] := 0.3083624;
   DATA[2205,34] := 2.0;
   DATA[2205,35] := 250.1602;
   DATA[2205,36] := 1.69801;
   DATA[2205,37] := 189.0861;
   DATA[2205,38] := 0.000128152;
   DATA[2205,39] := 1.0;
   DATA[2205,40] := 1.0;
   DATA[2206,0] := 2.617622;
   DATA[2206,1] := 864.542;
   DATA[2206,2] := 2.0;
   DATA[2206,3] := 2.0;
   DATA[2206,4] := 262.3686;
   DATA[2206,5] := 8.396116;
   DATA[2206,6] := 330.5563;
   DATA[2206,7] := 2.457694;
   DATA[2206,8] := 2.0;
   DATA[2206,9] := 2.0;
   DATA[2206,10] := 2.0;
   DATA[2206,11] := 19.73878;
   DATA[2206,12] := 2.209013;
   DATA[2206,13] := 811.3304;
   DATA[2206,14] := 1.0;
   DATA[2206,15] := 2.0;
   DATA[2206,16] := 1.0;
   DATA[2206,17] := 1.0;
   DATA[2206,18] := 1.0;
   DATA[2206,19] := 2.0;
   DATA[2206,20] := 148.808;
   DATA[2206,21] := 154.909;
   DATA[2206,22] := 1.71608;
   DATA[2206,23] := 845.2448;
   DATA[2206,24] := 2.0;
   DATA[2206,25] := 2.0;
   DATA[2206,26] := 7.873815;
   DATA[2206,27] := 143.9887;
   DATA[2206,28] := 261.8559;
   DATA[2206,29] := 12.03538;
   DATA[2206,30] := 1.724942;
   DATA[2206,31] := 1.296016;
   DATA[2206,32] := 0.7352687;
   DATA[2206,33] := 0.3083624;
   DATA[2206,34] := 2.0;
   DATA[2206,35] := 250.1602;
   DATA[2206,36] := 1.69801;
   DATA[2206,37] := 189.0861;
   DATA[2206,38] := 0.000128152;
   DATA[2206,39] := 1.0;
   DATA[2206,40] := 1.0;
   DATA[2207,0] := 2.607693;
   DATA[2207,1] := 864.2672;
   DATA[2207,2] := 2.0;
   DATA[2207,3] := 2.0;
   DATA[2207,4] := 262.3686;
   DATA[2207,5] := 8.396116;
   DATA[2207,6] := 330.5563;
   DATA[2207,7] := 2.458719;
   DATA[2207,8] := 2.0;
   DATA[2207,9] := 2.0;
   DATA[2207,10] := 2.0;
   DATA[2207,11] := 19.81881;
   DATA[2207,12] := 2.209013;
   DATA[2207,13] := 811.5307;
   DATA[2207,14] := 1.0;
   DATA[2207,15] := 2.0;
   DATA[2207,16] := 1.0;
   DATA[2207,17] := 1.0;
   DATA[2207,18] := 1.0;
   DATA[2207,19] := 2.0;
   DATA[2207,20] := 148.808;
   DATA[2207,21] := 154.909;
   DATA[2207,22] := 1.714798;
   DATA[2207,23] := 845.4371;
   DATA[2207,24] := 2.0;
   DATA[2207,25] := 2.0;
   DATA[2207,26] := 7.873815;
   DATA[2207,27] := 143.9887;
   DATA[2207,28] := 261.8559;
   DATA[2207,29] := 12.03538;
   DATA[2207,30] := 1.724942;
   DATA[2207,31] := 1.30178;
   DATA[2207,32] := 0.7352687;
   DATA[2207,33] := 0.3083624;
   DATA[2207,34] := 2.0;
   DATA[2207,35] := 250.1602;
   DATA[2207,36] := 1.69801;
   DATA[2207,37] := 189.0861;
   DATA[2207,38] := 0.000128152;
   DATA[2207,39] := 1.0;
   DATA[2207,40] := 1.0;
   DATA[2208,0] := 2.591679;
   DATA[2208,1] := 863.9532;
   DATA[2208,2] := 2.0;
   DATA[2208,3] := 2.0;
   DATA[2208,4] := 262.3686;
   DATA[2208,5] := 8.396116;
   DATA[2208,6] := 330.5563;
   DATA[2208,7] := 2.458976;
   DATA[2208,8] := 2.0;
